// ---- DUTs/IO/PDOs/DRV_Target_position_05240F14.TcDUT
{attribute 'GeneratedUsingTerminal: EL7211-0010-0032'}
{attribute addProperty BoxType "EL7211-0010-0032"}
{attribute addProperty Id "Target_positionAT %Q*UDINT4"}
{attribute addProperty CRC "86249236"}
{attribute addProperty Size "4"}
TYPE DRV_Target_position_05240F14 EXTENDS TcoIo.OutputBase_10CEE7DE :
STRUCT
    {attribute addProperty Name "Target_position"}
    Target_position AT %Q* : UDINT;
END_STRUCT
END_TYPE

// ---- DUTs/IO/PDOs/InfoData_433F0777.TcDUT
{attribute 'GeneratedUsingTerminal: EL7211-0010-0032'}
{attribute addProperty BoxType "EL7211-0010-0032"}
{attribute addProperty Id "AdsAddrAT %I*TcoIo.TcoAmsAddr0DcOutputShiftAT %I*DINT4DcInputShiftAT %I*DINT4Chn0AT %I*USINT1Chn1AT %I*USINT1StateAT %I*UINT2"}
{attribute addProperty CRC "1128204151"}
{attribute addProperty Size "12"}
TYPE InfoData_433F0777 EXTENDS TcoIo.InputBase_8311D824 :
STRUCT
    {attribute addProperty Name "AdsAddr"}
    AdsAddr AT %I* : TcoIo.TcoAmsAddr;
    {attribute addProperty Name "DcOutputShift"}
    DcOutputShift AT %I* : DINT;
    {attribute addProperty Name "DcInputShift"}
    DcInputShift AT %I* : DINT;
    {attribute addProperty Name "Chn0"}
    Chn0 AT %I* : USINT;
    {attribute addProperty Name "Chn1"}
    Chn1 AT %I* : USINT;
    {attribute addProperty Name "State"}
    State AT %I* : UINT;
END_STRUCT
END_TYPE

// ---- DUTs/IO/PDOs/SAI_Inputs_Channel_9DCD6557.TcDUT
{attribute 'GeneratedUsingTerminal: EL3692-0000-0020'}
{attribute addProperty BoxType "EL3692-0000-0020"}
{attribute addProperty Id "StatusAT %I*Status_439F40C310ValueAT %I*DINT4"}
{attribute addProperty CRC "2647483735"}
{attribute addProperty Size "14"}
TYPE SAI_Inputs_Channel_9DCD6557 EXTENDS TcoIo.InputBase_8311D824 :
STRUCT
    {attribute addProperty Name "Status"}
    Status AT %I* : Status_439F40C3;
    {attribute addProperty Name "Value"}
    Value AT %I* : DINT;
END_STRUCT
END_TYPE

// ---- DUTs/IO/PDOs/SAI_Range_Channel_BDBF6DA9.TcDUT
{attribute 'GeneratedUsingTerminal: EL3692-0000-0020'}
{attribute addProperty BoxType "EL3692-0000-0020"}
{attribute addProperty Id "SettingsAT %I*Settings_24C049402"}
{attribute addProperty CRC "3183439273"}
{attribute addProperty Size "2"}
TYPE SAI_Range_Channel_BDBF6DA9 EXTENDS TcoIo.InputBase_8311D824 :
STRUCT
    {attribute addProperty Name "Settings"}
    Settings AT %I* : Settings_24C04940;
END_STRUCT
END_TYPE

// ---- DUTs/IO/PDOs/SAI_Inputs_Real_Channel_CCECF13D.TcDUT
{attribute 'GeneratedUsingTerminal: EL3692-0000-0020'}
{attribute addProperty BoxType "EL3692-0000-0020"}
{attribute addProperty Id "ValueAT %I*REAL4"}
{attribute addProperty CRC "3438080317"}
{attribute addProperty Size "4"}
TYPE SAI_Inputs_Real_Channel_CCECF13D EXTENDS TcoIo.InputBase_8311D824 :
STRUCT
    {attribute addProperty Name "Value"}
    Value AT %I* : REAL;
END_STRUCT
END_TYPE

// ---- DUTs/IO/PDOs/SAI_Range_Control_Channel_F5D9BC22.TcDUT
{attribute 'GeneratedUsingTerminal: EL3692-0000-0020'}
{attribute addProperty BoxType "EL3692-0000-0020"}
{attribute addProperty Id "ControlAT %Q*Control_E49DBA1B4"}
{attribute addProperty CRC "4124687394"}
{attribute addProperty Size "4"}
TYPE SAI_Range_Control_Channel_F5D9BC22 EXTENDS TcoIo.OutputBase_10CEE7DE :
STRUCT
    {attribute addProperty Name "Control"}
    Control AT %Q* : Control_E49DBA1B;
END_STRUCT
END_TYPE

// ---- DUTs/IO/PDOs/In_389F2F15.TcDUT
{attribute 'GeneratedUsingTerminal: Flexi Soft EtherCAT Gateway-0000-0001'}
{attribute addProperty BoxType "Flexi Soft EtherCAT Gateway-0000-0001"}
{attribute addProperty Id "DiagAT %I*USINT1In_Dataset1AT %I*ARRAY [0..9] OF BYTE0In_Dataset2AT %I*ARRAY [0..9] OF BYTE0In_Dataset3AT %I*ARRAY [0..9] OF BYTE0In_Dataset4AT %I*ARRAY [0..9] OF BYTE0In_Dataset5AT %I*ARRAY [0..9] OF BYTE0"}
{attribute addProperty CRC "949956373"}
{attribute addProperty Size "1"}
TYPE In_389F2F15 EXTENDS TcoIo.InputBase_8311D824 :
STRUCT
    {attribute addProperty Name "Diag"}
    Diag AT %I* : USINT;
    {attribute addProperty Name "In_Dataset1"}
    In_Dataset1 AT %I* : ARRAY[0..9] OF BYTE;
    {attribute addProperty Name "In_Dataset2"}
    In_Dataset2 AT %I* : ARRAY[0..9] OF BYTE;
    {attribute addProperty Name "In_Dataset3"}
    In_Dataset3 AT %I* : ARRAY[0..9] OF BYTE;
    {attribute addProperty Name "In_Dataset4"}
    In_Dataset4 AT %I* : ARRAY[0..9] OF BYTE;
    {attribute addProperty Name "In_Dataset5"}
    In_Dataset5 AT %I* : ARRAY[0..9] OF BYTE;
END_STRUCT
END_TYPE

// ---- DUTs/IO/PDOs/Out_81AAEF2D.TcDUT
{attribute 'GeneratedUsingTerminal: Flexi Soft EtherCAT Gateway-0000-0001'}
{attribute addProperty BoxType "Flexi Soft EtherCAT Gateway-0000-0001"}
{attribute addProperty Id "Out_Dataset1AT %Q*ARRAY [0..9] OF BYTE0Out_Dataset2AT %Q*ARRAY [0..9] OF BYTE0Out_Dataset3AT %Q*ARRAY [0..9] OF BYTE0Out_Dataset4AT %Q*ARRAY [0..9] OF BYTE0Out_Dataset5AT %Q*ARRAY [0..9] OF BYTE0"}
{attribute addProperty CRC "2175463213"}
{attribute addProperty Size "0"}
TYPE Out_81AAEF2D EXTENDS TcoIo.OutputBase_10CEE7DE :
STRUCT
    {attribute addProperty Name "Out_Dataset1"}
    Out_Dataset1 AT %Q* : ARRAY[0..9] OF BYTE;
    {attribute addProperty Name "Out_Dataset2"}
    Out_Dataset2 AT %Q* : ARRAY[0..9] OF BYTE;
    {attribute addProperty Name "Out_Dataset3"}
    Out_Dataset3 AT %Q* : ARRAY[0..9] OF BYTE;
    {attribute addProperty Name "Out_Dataset4"}
    Out_Dataset4 AT %Q* : ARRAY[0..9] OF BYTE;
    {attribute addProperty Name "Out_Dataset5"}
    Out_Dataset5 AT %Q* : ARRAY[0..9] OF BYTE;
END_STRUCT
END_TYPE

// ---- DUTs/IO/PDOs/ENC_Status_compact_4D066E1A.TcDUT
{attribute 'GeneratedUsingTerminal: EL7041-1000-0021'}
{attribute addProperty BoxType "EL7041-1000-0021"}
{attribute addProperty Id "StatusAT %I*Status_8CBE219F12Counter_valueAT %I*UINT2Latch_valueAT %I*UINT2"}
{attribute addProperty CRC "1292267034"}
{attribute addProperty Size "16"}
TYPE ENC_Status_compact_4D066E1A EXTENDS TcoIo.InputBase_8311D824 :
STRUCT
    {attribute addProperty Name "Status"}
    Status AT %I* : Status_8CBE219F;
    {attribute addProperty Name "Counter_value"}
    Counter_value AT %I* : UINT;
    {attribute addProperty Name "Latch_value"}
    Latch_value AT %I* : UINT;
END_STRUCT
END_TYPE

// ---- DUTs/IO/PDOs/STM_Status_36ED096F.TcDUT
{attribute 'GeneratedUsingTerminal: EL7041-1000-0021'}
{attribute addProperty BoxType "EL7041-1000-0021"}
{attribute addProperty Id "StatusAT %I*Status_B679584511"}
{attribute addProperty CRC "921504111"}
{attribute addProperty Size "11"}
TYPE STM_Status_36ED096F EXTENDS TcoIo.InputBase_8311D824 :
STRUCT
    {attribute addProperty Name "Status"}
    Status AT %I* : Status_B6795845;
END_STRUCT
END_TYPE

// ---- DUTs/IO/PDOs/ENC_Control_compact_21E2D14D.TcDUT
{attribute 'GeneratedUsingTerminal: EL7041-1000-0021'}
{attribute addProperty BoxType "EL7041-1000-0021"}
{attribute addProperty Id "ControlAT %Q*Control_6EF2C5D04Set_counter_valueAT %Q*UINT2"}
{attribute addProperty CRC "568512845"}
{attribute addProperty Size "6"}
TYPE ENC_Control_compact_21E2D14D EXTENDS TcoIo.OutputBase_10CEE7DE :
STRUCT
    {attribute addProperty Name "Control"}
    Control AT %Q* : Control_6EF2C5D0;
    {attribute addProperty Name "Set_counter_value"}
    Set_counter_value AT %Q* : UINT;
END_STRUCT
END_TYPE

// ---- DUTs/IO/PDOs/STM_Control_5A8B5016.TcDUT
{attribute 'GeneratedUsingTerminal: EL7041-1000-0021'}
{attribute addProperty BoxType "EL7041-1000-0021"}
{attribute addProperty Id "ControlAT %Q*Control_C948E0F23"}
{attribute addProperty CRC "1519079446"}
{attribute addProperty Size "3"}
TYPE STM_Control_5A8B5016 EXTENDS TcoIo.OutputBase_10CEE7DE :
STRUCT
    {attribute addProperty Name "Control"}
    Control AT %Q* : Control_C948E0F2;
END_STRUCT
END_TYPE

// ---- DUTs/IO/PDOs/STM_Velocity_A47A3F41.TcDUT
{attribute 'GeneratedUsingTerminal: EL7041-1000-0021'}
{attribute addProperty BoxType "EL7041-1000-0021"}
{attribute addProperty Id "VelocityAT %Q*INT2"}
{attribute addProperty CRC "2759475009"}
{attribute addProperty Size "2"}
TYPE STM_Velocity_A47A3F41 EXTENDS TcoIo.OutputBase_10CEE7DE :
STRUCT
    {attribute addProperty Name "Velocity"}
    Velocity AT %Q* : INT;
END_STRUCT
END_TYPE

// ---- DUTs/IO/PDOs/InfoData_D50C8545.TcDUT
{attribute 'GeneratedUsingTerminal: EL7041-1000-0021'}
{attribute addProperty BoxType "EL7041-1000-0021"}
{attribute addProperty Id "AdsAddrAT %I*TcoIo.TcoAmsAddr0Chn0AT %I*USINT1StateAT %I*UINT2"}
{attribute addProperty CRC "3574367557"}
{attribute addProperty Size "3"}
TYPE InfoData_D50C8545 EXTENDS TcoIo.InputBase_8311D824 :
STRUCT
    {attribute addProperty Name "AdsAddr"}
    AdsAddr AT %I* : TcoIo.TcoAmsAddr;
    {attribute addProperty Name "Chn0"}
    Chn0 AT %I* : USINT;
    {attribute addProperty Name "State"}
    State AT %I* : UINT;
END_STRUCT
END_TYPE

// ---- DUTs/IO/PDOs/AT_x_26CC547D.TcDUT
{attribute 'GeneratedUsingTerminal: IndraDrive MPB20-0003-0000'}
{attribute addProperty BoxType "IndraDrive MPB20-0003-0000"}
{attribute addProperty Id "Drive_status_wordAT %I*UINT2Position_feedback_value_1AT %I*DINT4"}
{attribute addProperty CRC "650925181"}
{attribute addProperty Size "6"}
TYPE AT_x_26CC547D EXTENDS TcoIo.InputBase_8311D824 :
STRUCT
    {attribute addProperty Name "Drive_status_word"}
    Drive_status_word AT %I* : UINT;
    {attribute addProperty Name "Position_feedback_value_1"}
    Position_feedback_value_1 AT %I* : DINT;
END_STRUCT
END_TYPE

// ---- DUTs/IO/Boxes/EK1200_013D0B49.TcDUT
{attribute 'GeneratedUsingTerminal: EK1200-1388-0000'}
{attribute addProperty VendorId "#x00000002"}
{attribute addProperty BoxType "EK1200-1388-0000"}
{attribute addProperty Description "EK1200-5000 EtherCAT Power supply (2A E-Bus)"}
{attribute addProperty Physics "YK"}
{attribute addProperty Id "EK1200"}
{attribute addProperty CRC "20777801"}
{attribute addProperty Size "0"}
TYPE EK1200_013D0B49 EXTENDS TcoIo.EtcSlaveBoxBase_77A0E4A7 :
STRUCT
END_STRUCT
END_TYPE

// ---- DUTs/IO/Boxes/EL6002_CD897635.TcDUT
{attribute 'GeneratedUsingTerminal: EL6002-0000-0019'}
{attribute addProperty VendorId "#x00000002"}
{attribute addProperty BoxType "EL6002-0000-0019"}
{attribute addProperty Description "EL6002 Interface 2Ch. (RS232)"}
{attribute addProperty Physics "KK"}
{attribute addProperty Id "COM_TxPDO_Map_Inputs_Channel_1AT %I*COM_TxPDO_Map_Inputs_Channel_3801C95E30COM_TxPDO_Map_Inputs_Channel_2AT %I*COM_TxPDO_Map_Inputs_Channel_3801C95E30COM_RxPDO_Map_Outputs_Channel_1AT %Q*COM_RxPDO_Map_Outputs_Channel_EADA2E0D27COM_RxPDO_Map_Outputs_Channel_2AT %Q*COM_RxPDO_Map_Outputs_Channel_EADA2E0D27WcStateAT %I*WcState_9091E0EB2InfoDataAT %I*InfoData_23CBA8372"}
{attribute addProperty CRC "3448337973"}
{attribute addProperty Size "118"}
TYPE EL6002_CD897635 EXTENDS TcoIo.EtcSlaveTerminalBase_947E5A46 :
STRUCT
    {attribute addProperty Name "COM_TxPDO_Map_Inputs_Channel_1"}
    COM_TxPDO_Map_Inputs_Channel_1 : COM_TxPDO_Map_Inputs_Channel_3801C95E;
    {attribute addProperty Name "COM_TxPDO_Map_Inputs_Channel_2"}
    COM_TxPDO_Map_Inputs_Channel_2 : COM_TxPDO_Map_Inputs_Channel_3801C95E;
    {attribute addProperty Name "COM_RxPDO_Map_Outputs_Channel_1"}
    COM_RxPDO_Map_Outputs_Channel_1 : COM_RxPDO_Map_Outputs_Channel_EADA2E0D;
    {attribute addProperty Name "COM_RxPDO_Map_Outputs_Channel_2"}
    COM_RxPDO_Map_Outputs_Channel_2 : COM_RxPDO_Map_Outputs_Channel_EADA2E0D;
    {attribute addProperty Name "WcState"}
    WcState : TcoIo.WcState_9091E0EB;
    {attribute addProperty Name "InfoData"}
    InfoData : TcoIo.InfoData_23CBA837;
END_STRUCT
END_TYPE

// ---- DUTs/IO/Boxes/EL1809_32157CFD.TcDUT
{attribute 'GeneratedUsingTerminal: EL1809-0000-0018'}
{attribute addProperty VendorId "#x00000002"}
{attribute addProperty BoxType "EL1809-0000-0018"}
{attribute addProperty Description "EL1809 16Ch. Dig. Input 24V, 3ms"}
{attribute addProperty Physics "KK"}
{attribute addProperty Id "Channel_1AT %I*Channel_830843C11Channel_2AT %I*Channel_830843C11Channel_3AT %I*Channel_830843C11Channel_4AT %I*Channel_830843C11Channel_5AT %I*Channel_830843C11Channel_6AT %I*Channel_830843C11Channel_7AT %I*Channel_830843C11Channel_8AT %I*Channel_830843C11Channel_9AT %I*Channel_830843C11Channel_10AT %I*Channel_830843C11Channel_11AT %I*Channel_830843C11Channel_12AT %I*Channel_830843C11Channel_13AT %I*Channel_830843C11Channel_14AT %I*Channel_830843C11Channel_15AT %I*Channel_830843C11Channel_16AT %I*Channel_830843C11WcStateAT %I*WcState_9091E0EB2InfoDataAT %I*InfoData_6F19DB2B2"}
{attribute addProperty CRC "840269053"}
{attribute addProperty Size "20"}
TYPE EL1809_32157CFD EXTENDS TcoIo.EtcSlaveTerminalBase_947E5A46 :
STRUCT
    {attribute addProperty Name "Channel_1"}
    Channel_1 : Channel_830843C1;
    {attribute addProperty Name "Channel_2"}
    Channel_2 : Channel_830843C1;
    {attribute addProperty Name "Channel_3"}
    Channel_3 : Channel_830843C1;
    {attribute addProperty Name "Channel_4"}
    Channel_4 : Channel_830843C1;
    {attribute addProperty Name "Channel_5"}
    Channel_5 : Channel_830843C1;
    {attribute addProperty Name "Channel_6"}
    Channel_6 : Channel_830843C1;
    {attribute addProperty Name "Channel_7"}
    Channel_7 : Channel_830843C1;
    {attribute addProperty Name "Channel_8"}
    Channel_8 : Channel_830843C1;
    {attribute addProperty Name "Channel_9"}
    Channel_9 : Channel_830843C1;
    {attribute addProperty Name "Channel_10"}
    Channel_10 : Channel_830843C1;
    {attribute addProperty Name "Channel_11"}
    Channel_11 : Channel_830843C1;
    {attribute addProperty Name "Channel_12"}
    Channel_12 : Channel_830843C1;
    {attribute addProperty Name "Channel_13"}
    Channel_13 : Channel_830843C1;
    {attribute addProperty Name "Channel_14"}
    Channel_14 : Channel_830843C1;
    {attribute addProperty Name "Channel_15"}
    Channel_15 : Channel_830843C1;
    {attribute addProperty Name "Channel_16"}
    Channel_16 : Channel_830843C1;
    {attribute addProperty Name "WcState"}
    WcState : TcoIo.WcState_9091E0EB;
    {attribute addProperty Name "InfoData"}
    InfoData : TcoIo.InfoData_6F19DB2B;
END_STRUCT
END_TYPE

// ---- DUTs/IO/Boxes/EL2809_2B6483BD.TcDUT
{attribute 'GeneratedUsingTerminal: EL2809-0000-0018'}
{attribute addProperty VendorId "#x00000002"}
{attribute addProperty BoxType "EL2809-0000-0018"}
{attribute addProperty Description "EL2809 16Ch. Dig. Output 24V, 0.5A"}
{attribute addProperty Physics "KK"}
{attribute addProperty Id "Channel_1AT %Q*Channel_42CA91F71Channel_2AT %Q*Channel_42CA91F71Channel_3AT %Q*Channel_42CA91F71Channel_4AT %Q*Channel_42CA91F71Channel_5AT %Q*Channel_42CA91F71Channel_6AT %Q*Channel_42CA91F71Channel_7AT %Q*Channel_42CA91F71Channel_8AT %Q*Channel_42CA91F71Channel_9AT %Q*Channel_42CA91F71Channel_10AT %Q*Channel_42CA91F71Channel_11AT %Q*Channel_42CA91F71Channel_12AT %Q*Channel_42CA91F71Channel_13AT %Q*Channel_42CA91F71Channel_14AT %Q*Channel_42CA91F71Channel_15AT %Q*Channel_42CA91F71Channel_16AT %Q*Channel_42CA91F71WcStateAT %I*WcState_0B2B16F91InfoDataAT %I*InfoData_6F19DB2B2"}
{attribute addProperty CRC "728007613"}
{attribute addProperty Size "19"}
TYPE EL2809_2B6483BD EXTENDS TcoIo.EtcSlaveTerminalBase_947E5A46 :
STRUCT
    {attribute addProperty Name "Channel_1"}
    Channel_1 : Channel_42CA91F7;
    {attribute addProperty Name "Channel_2"}
    Channel_2 : Channel_42CA91F7;
    {attribute addProperty Name "Channel_3"}
    Channel_3 : Channel_42CA91F7;
    {attribute addProperty Name "Channel_4"}
    Channel_4 : Channel_42CA91F7;
    {attribute addProperty Name "Channel_5"}
    Channel_5 : Channel_42CA91F7;
    {attribute addProperty Name "Channel_6"}
    Channel_6 : Channel_42CA91F7;
    {attribute addProperty Name "Channel_7"}
    Channel_7 : Channel_42CA91F7;
    {attribute addProperty Name "Channel_8"}
    Channel_8 : Channel_42CA91F7;
    {attribute addProperty Name "Channel_9"}
    Channel_9 : Channel_42CA91F7;
    {attribute addProperty Name "Channel_10"}
    Channel_10 : Channel_42CA91F7;
    {attribute addProperty Name "Channel_11"}
    Channel_11 : Channel_42CA91F7;
    {attribute addProperty Name "Channel_12"}
    Channel_12 : Channel_42CA91F7;
    {attribute addProperty Name "Channel_13"}
    Channel_13 : Channel_42CA91F7;
    {attribute addProperty Name "Channel_14"}
    Channel_14 : Channel_42CA91F7;
    {attribute addProperty Name "Channel_15"}
    Channel_15 : Channel_42CA91F7;
    {attribute addProperty Name "Channel_16"}
    Channel_16 : Channel_42CA91F7;
    {attribute addProperty Name "WcState"}
    WcState : TcoIo.WcState_0B2B16F9;
    {attribute addProperty Name "InfoData"}
    InfoData : TcoIo.InfoData_6F19DB2B;
END_STRUCT
END_TYPE

// ---- DUTs/IO/Boxes/EL4004_E203F875.TcDUT
{attribute 'GeneratedUsingTerminal: EL4004-0000-0020'}
{attribute addProperty VendorId "#x00000002"}
{attribute addProperty BoxType "EL4004-0000-0020"}
{attribute addProperty Description "EL4004 4Ch. Ana. Output 0-10V, 12bit"}
{attribute addProperty Physics "KK"}
{attribute addProperty Id "AO_Outputs_Channel_1AT %Q*AO_Output_Channel_BA7EBB7C2AO_Outputs_Channel_2AT %Q*AO_Output_Channel_BA7EBB7C2AO_Outputs_Channel_3AT %Q*AO_Output_Channel_BA7EBB7C2AO_Outputs_Channel_4AT %Q*AO_Output_Channel_BA7EBB7C2WcStateAT %I*WcState_0B2B16F91InfoDataAT %I*InfoData_23CBA8372"}
{attribute addProperty CRC "3791911029"}
{attribute addProperty Size "11"}
TYPE EL4004_E203F875 EXTENDS TcoIo.EtcSlaveTerminalBase_947E5A46 :
STRUCT
    {attribute addProperty Name "AO_Outputs_Channel_1"}
    AO_Outputs_Channel_1 : AO_Output_Channel_BA7EBB7C;
    {attribute addProperty Name "AO_Outputs_Channel_2"}
    AO_Outputs_Channel_2 : AO_Output_Channel_BA7EBB7C;
    {attribute addProperty Name "AO_Outputs_Channel_3"}
    AO_Outputs_Channel_3 : AO_Output_Channel_BA7EBB7C;
    {attribute addProperty Name "AO_Outputs_Channel_4"}
    AO_Outputs_Channel_4 : AO_Output_Channel_BA7EBB7C;
    {attribute addProperty Name "WcState"}
    WcState : TcoIo.WcState_0B2B16F9;
    {attribute addProperty Name "InfoData"}
    InfoData : TcoIo.InfoData_23CBA837;
END_STRUCT
END_TYPE

// ---- DUTs/IO/Boxes/EL6001_0DE01E7E.TcDUT
{attribute 'GeneratedUsingTerminal: EL6001-0000-0020'}
{attribute addProperty VendorId "#x00000002"}
{attribute addProperty BoxType "EL6001-0000-0020"}
{attribute addProperty Description "EL6001 Interface (RS232)"}
{attribute addProperty Physics "KK"}
{attribute addProperty Id "COM_InputsAT %I*COM_Inputs_3801C95E30COM_OutputsAT %Q*COM_Outputs_DEF408EC27WcStateAT %I*WcState_9091E0EB2InfoDataAT %I*InfoData_23CBA8372"}
{attribute addProperty CRC "232791678"}
{attribute addProperty Size "61"}
TYPE EL6001_0DE01E7E EXTENDS TcoIo.EtcSlaveTerminalBase_947E5A46 :
STRUCT
    {attribute addProperty Name "COM_Inputs"}
    COM_Inputs : COM_Inputs_3801C95E;
    {attribute addProperty Name "COM_Outputs"}
    COM_Outputs : COM_Outputs_DEF408EC;
    {attribute addProperty Name "WcState"}
    WcState : TcoIo.WcState_9091E0EB;
    {attribute addProperty Name "InfoData"}
    InfoData : TcoIo.InfoData_23CBA837;
END_STRUCT
END_TYPE

// ---- DUTs/IO/Boxes/EL9011_D65D3D32.TcDUT
{attribute 'GeneratedUsingTerminal: EL9011--0000'}
{attribute addProperty VendorId "#x00000002"}
{attribute addProperty BoxType "EL9011--0000"}
{attribute addProperty Description "EL9011 End Terminal"}
{attribute addProperty Physics ""}
{attribute addProperty Id "EL9011"}
{attribute addProperty CRC "3596434738"}
{attribute addProperty Size "0"}
TYPE EL9011_D65D3D32 EXTENDS TcoIo.EtcSlaveEndTerminalBase_866C7F0C :
STRUCT
END_STRUCT
END_TYPE

// ---- DUTs/IO/Boxes/EK1100_1FC0878B.TcDUT
{attribute 'GeneratedUsingTerminal: EK1100-0000-0018'}
{attribute addProperty VendorId "#x00000002"}
{attribute addProperty BoxType "EK1100-0000-0018"}
{attribute addProperty Description "EK1100 EtherCAT Coupler (2A E-Bus)"}
{attribute addProperty Physics "YKY"}
{attribute addProperty Id "InfoDataAT %I*InfoData_6F19DB2B2"}
{attribute addProperty CRC "532711307"}
{attribute addProperty Size "2"}
TYPE EK1100_1FC0878B EXTENDS TcoIo.EtcSlaveBoxBase_77A0E4A7 :
STRUCT
    {attribute addProperty Name "InfoData"}
    InfoData : TcoIo.InfoData_6F19DB2B;
END_STRUCT
END_TYPE

// ---- DUTs/IO/Boxes/EK1122_1FC0878B.TcDUT
{attribute 'GeneratedUsingTerminal: EK1122-0000-0018'}
{attribute addProperty VendorId "#x00000002"}
{attribute addProperty BoxType "EK1122-0000-0018"}
{attribute addProperty Description "EK1122 2 port EtherCAT junction"}
{attribute addProperty Physics "KYKY"}
{attribute addProperty Id "InfoDataAT %I*InfoData_6F19DB2B2"}
{attribute addProperty CRC "532711307"}
{attribute addProperty Size "2"}
TYPE EK1122_1FC0878B EXTENDS TcoIo.EtcSlaveTerminalBase_947E5A46 :
STRUCT
    {attribute addProperty Name "InfoData"}
    InfoData : TcoIo.InfoData_6F19DB2B;
END_STRUCT
END_TYPE

// ---- DUTs/IO/Boxes/EL3174_B71BFF42.TcDUT
{attribute 'GeneratedUsingTerminal: EL3174-0002-0017'}
{attribute addProperty VendorId "#x00000002"}
{attribute addProperty BoxType "EL3174-0002-0017"}
{attribute addProperty Description "EL3174-0002 4Ch. Ana. Input +/-10V, +/-20mA 16 Bit, Isolated Channels"}
{attribute addProperty Physics "KK"}
{attribute addProperty Id "AI_Standard_Channel_1AT %I*AI_Standard_Channel_A8DF64E310AI_Standard_Channel_2AT %I*AI_Standard_Channel_A8DF64E310AI_Standard_Channel_3AT %I*AI_Standard_Channel_A8DF64E310AI_Standard_Channel_4AT %I*AI_Standard_Channel_A8DF64E310WcStateAT %I*WcState_9091E0EB2InfoDataAT %I*InfoData_23CBA8372"}
{attribute addProperty CRC "3072065346"}
{attribute addProperty Size "44"}
TYPE EL3174_B71BFF42 EXTENDS TcoIo.EtcSlaveTerminalBase_947E5A46 :
STRUCT
    {attribute addProperty Name "AI_Standard_Channel_1"}
    AI_Standard_Channel_1 : AI_Standard_Channel_A8DF64E3;
    {attribute addProperty Name "AI_Standard_Channel_2"}
    AI_Standard_Channel_2 : AI_Standard_Channel_A8DF64E3;
    {attribute addProperty Name "AI_Standard_Channel_3"}
    AI_Standard_Channel_3 : AI_Standard_Channel_A8DF64E3;
    {attribute addProperty Name "AI_Standard_Channel_4"}
    AI_Standard_Channel_4 : AI_Standard_Channel_A8DF64E3;
    {attribute addProperty Name "WcState"}
    WcState : TcoIo.WcState_9091E0EB;
    {attribute addProperty Name "InfoData"}
    InfoData : TcoIo.InfoData_23CBA837;
END_STRUCT
END_TYPE

// ---- DUTs/IO/Boxes/EL3011_7A495228.TcDUT
{attribute 'GeneratedUsingTerminal: EL3011-0000-0018'}
{attribute addProperty VendorId "#x00000002"}
{attribute addProperty BoxType "EL3011-0000-0018"}
{attribute addProperty Description "EL3011 4Ch. Ana. Input 0-20mA DIFF"}
{attribute addProperty Physics "KK"}
{attribute addProperty Id "AI_StandardAT %I*AI_Standard_Channel_4A3944819WcStateAT %I*WcState_9091E0EB2InfoDataAT %I*InfoData_23CBA8372"}
{attribute addProperty CRC "2051625512"}
{attribute addProperty Size "13"}
TYPE EL3011_7A495228 EXTENDS TcoIo.EtcSlaveTerminalBase_947E5A46 :
STRUCT
    {attribute addProperty Name "AI_Standard"}
    AI_Standard : AI_Standard_Channel_4A394481;
    {attribute addProperty Name "WcState"}
    WcState : TcoIo.WcState_9091E0EB;
    {attribute addProperty Name "InfoData"}
    InfoData : TcoIo.InfoData_23CBA837;
END_STRUCT
END_TYPE

// ---- DUTs/IO/Boxes/EL2008_E2806B95.TcDUT
{attribute 'GeneratedUsingTerminal: EL2008-0000-0017'}
{attribute addProperty VendorId "#x00000002"}
{attribute addProperty BoxType "EL2008-0000-0017"}
{attribute addProperty Description "EL2008 8Ch. Dig. Output 24V, 0.5A"}
{attribute addProperty Physics "KK"}
{attribute addProperty Id "Channel_1AT %Q*Channel_42CA91F71Channel_2AT %Q*Channel_42CA91F71Channel_3AT %Q*Channel_42CA91F71Channel_4AT %Q*Channel_42CA91F71Channel_5AT %Q*Channel_42CA91F71Channel_6AT %Q*Channel_42CA91F71Channel_7AT %Q*Channel_42CA91F71Channel_8AT %Q*Channel_42CA91F71WcStateAT %I*WcState_0B2B16F91InfoDataAT %I*InfoData_6F19DB2B2"}
{attribute addProperty CRC "3800066965"}
{attribute addProperty Size "11"}
TYPE EL2008_E2806B95 EXTENDS TcoIo.EtcSlaveTerminalBase_947E5A46 :
STRUCT
    {attribute addProperty Name "Channel_1"}
    Channel_1 : Channel_42CA91F7;
    {attribute addProperty Name "Channel_2"}
    Channel_2 : Channel_42CA91F7;
    {attribute addProperty Name "Channel_3"}
    Channel_3 : Channel_42CA91F7;
    {attribute addProperty Name "Channel_4"}
    Channel_4 : Channel_42CA91F7;
    {attribute addProperty Name "Channel_5"}
    Channel_5 : Channel_42CA91F7;
    {attribute addProperty Name "Channel_6"}
    Channel_6 : Channel_42CA91F7;
    {attribute addProperty Name "Channel_7"}
    Channel_7 : Channel_42CA91F7;
    {attribute addProperty Name "Channel_8"}
    Channel_8 : Channel_42CA91F7;
    {attribute addProperty Name "WcState"}
    WcState : TcoIo.WcState_0B2B16F9;
    {attribute addProperty Name "InfoData"}
    InfoData : TcoIo.InfoData_6F19DB2B;
END_STRUCT
END_TYPE

// ---- DUTs/IO/Boxes/EK1110_1FC0878B.TcDUT
{attribute 'GeneratedUsingTerminal: EK1110-0000-0017'}
{attribute addProperty VendorId "#x00000002"}
{attribute addProperty BoxType "EK1110-0000-0017"}
{attribute addProperty Description "EK1110 EtherCAT extension"}
{attribute addProperty Physics "KY"}
{attribute addProperty Id "InfoDataAT %I*InfoData_6F19DB2B2"}
{attribute addProperty CRC "532711307"}
{attribute addProperty Size "2"}
TYPE EK1110_1FC0878B EXTENDS TcoIo.EtcSlaveTerminalBase_947E5A46 :
STRUCT
    {attribute addProperty Name "InfoData"}
    InfoData : TcoIo.InfoData_6F19DB2B;
END_STRUCT
END_TYPE

// ---- DUTs/IO/Boxes/EL1819_32157CFD.TcDUT
{attribute 'GeneratedUsingTerminal: EL1819-0000-0018'}
{attribute addProperty VendorId "#x00000002"}
{attribute addProperty BoxType "EL1819-0000-0018"}
{attribute addProperty Description "EL1819 16Ch. Dig. Input 24V, 10Ã‚Âµs"}
{attribute addProperty Physics "KK"}
{attribute addProperty Id "Channel_1AT %I*Channel_830843C11Channel_2AT %I*Channel_830843C11Channel_3AT %I*Channel_830843C11Channel_4AT %I*Channel_830843C11Channel_5AT %I*Channel_830843C11Channel_6AT %I*Channel_830843C11Channel_7AT %I*Channel_830843C11Channel_8AT %I*Channel_830843C11Channel_9AT %I*Channel_830843C11Channel_10AT %I*Channel_830843C11Channel_11AT %I*Channel_830843C11Channel_12AT %I*Channel_830843C11Channel_13AT %I*Channel_830843C11Channel_14AT %I*Channel_830843C11Channel_15AT %I*Channel_830843C11Channel_16AT %I*Channel_830843C11WcStateAT %I*WcState_9091E0EB2InfoDataAT %I*InfoData_6F19DB2B2"}
{attribute addProperty CRC "840269053"}
{attribute addProperty Size "20"}
TYPE EL1819_32157CFD EXTENDS TcoIo.EtcSlaveTerminalBase_947E5A46 :
STRUCT
    {attribute addProperty Name "Channel_1"}
    Channel_1 : Channel_830843C1;
    {attribute addProperty Name "Channel_2"}
    Channel_2 : Channel_830843C1;
    {attribute addProperty Name "Channel_3"}
    Channel_3 : Channel_830843C1;
    {attribute addProperty Name "Channel_4"}
    Channel_4 : Channel_830843C1;
    {attribute addProperty Name "Channel_5"}
    Channel_5 : Channel_830843C1;
    {attribute addProperty Name "Channel_6"}
    Channel_6 : Channel_830843C1;
    {attribute addProperty Name "Channel_7"}
    Channel_7 : Channel_830843C1;
    {attribute addProperty Name "Channel_8"}
    Channel_8 : Channel_830843C1;
    {attribute addProperty Name "Channel_9"}
    Channel_9 : Channel_830843C1;
    {attribute addProperty Name "Channel_10"}
    Channel_10 : Channel_830843C1;
    {attribute addProperty Name "Channel_11"}
    Channel_11 : Channel_830843C1;
    {attribute addProperty Name "Channel_12"}
    Channel_12 : Channel_830843C1;
    {attribute addProperty Name "Channel_13"}
    Channel_13 : Channel_830843C1;
    {attribute addProperty Name "Channel_14"}
    Channel_14 : Channel_830843C1;
    {attribute addProperty Name "Channel_15"}
    Channel_15 : Channel_830843C1;
    {attribute addProperty Name "Channel_16"}
    Channel_16 : Channel_830843C1;
    {attribute addProperty Name "WcState"}
    WcState : TcoIo.WcState_9091E0EB;
    {attribute addProperty Name "InfoData"}
    InfoData : TcoIo.InfoData_6F19DB2B;
END_STRUCT
END_TYPE

// ---- DUTs/IO/Boxes/EL2788_E2806B95.TcDUT
{attribute 'GeneratedUsingTerminal: EL2788-0000-0016'}
{attribute addProperty VendorId "#x00000002"}
{attribute addProperty BoxType "EL2788-0000-0016"}
{attribute addProperty Description "EL2788 8Ch. Dig. Output 24V AC/DC, 2A"}
{attribute addProperty Physics "KK"}
{attribute addProperty Id "Channel_1AT %Q*Channel_42CA91F71Channel_2AT %Q*Channel_42CA91F71Channel_3AT %Q*Channel_42CA91F71Channel_4AT %Q*Channel_42CA91F71Channel_5AT %Q*Channel_42CA91F71Channel_6AT %Q*Channel_42CA91F71Channel_7AT %Q*Channel_42CA91F71Channel_8AT %Q*Channel_42CA91F71WcStateAT %I*WcState_0B2B16F91InfoDataAT %I*InfoData_6F19DB2B2"}
{attribute addProperty CRC "3800066965"}
{attribute addProperty Size "11"}
TYPE EL2788_E2806B95 EXTENDS TcoIo.EtcSlaveTerminalBase_947E5A46 :
STRUCT
    {attribute addProperty Name "Channel_1"}
    Channel_1 : Channel_42CA91F7;
    {attribute addProperty Name "Channel_2"}
    Channel_2 : Channel_42CA91F7;
    {attribute addProperty Name "Channel_3"}
    Channel_3 : Channel_42CA91F7;
    {attribute addProperty Name "Channel_4"}
    Channel_4 : Channel_42CA91F7;
    {attribute addProperty Name "Channel_5"}
    Channel_5 : Channel_42CA91F7;
    {attribute addProperty Name "Channel_6"}
    Channel_6 : Channel_42CA91F7;
    {attribute addProperty Name "Channel_7"}
    Channel_7 : Channel_42CA91F7;
    {attribute addProperty Name "Channel_8"}
    Channel_8 : Channel_42CA91F7;
    {attribute addProperty Name "WcState"}
    WcState : TcoIo.WcState_0B2B16F9;
    {attribute addProperty Name "InfoData"}
    InfoData : TcoIo.InfoData_6F19DB2B;
END_STRUCT
END_TYPE

// ---- DUTs/IO/Boxes/EL3773_F128CC82.TcDUT
{attribute 'GeneratedUsingTerminal: EL3773-0000-0021'}
{attribute addProperty VendorId "#x00000002"}
{attribute addProperty BoxType "EL3773-0000-0021"}
{attribute addProperty Description "EL3773 3 Ch. Power Monitoring, Oversample"}
{attribute addProperty Physics "KK"}
{attribute addProperty Id "L1_Voltage_StatusAT %I*L1_Voltage_Status_7371B0437L1_Voltage_SamplesAT %I*L1_Voltage_Samples_41AEB7FF20L1_Current_StatusAT %I*L1_Current_Status_82DECBF67L1_Current_SamplesAT %I*L1_Current_Samples_9EC08B3E20L2_Voltage_StatusAT %I*L2_Voltage_Status_0D1813FE7L2_Voltage_SamplesAT %I*L2_Voltage_Samples_75D833AF20L2_Current_StatusAT %I*L2_Current_Status_FCB7684B7L2_Current_SamplesAT %I*L2_Current_Samples_AAB60F6E20L3_Voltage_StatusAT %I*L3_Voltage_Status_273F72957L3_Voltage_SamplesAT %I*L3_Voltage_Samples_660A4F9F20L3_Current_StatusAT %I*L3_Current_Status_D69009207L3_Current_SamplesAT %I*L3_Current_Samples_B964735E20AI_NextSync1TimeAT %I*AI_NextSync1Time_6DC4D2968AI_Sample_CountAT %I*AI_Sample_Count_EA88CAD92WcStateAT %I*WcState_9091E0EB2InfoDataAT %I*InfoData_B84DBEC510"}
{attribute addProperty CRC "4045982850"}
{attribute addProperty Size "184"}
TYPE EL3773_F128CC82 EXTENDS TcoIo.EtcSlaveTerminalBase_947E5A46 :
STRUCT
    {attribute addProperty Name "L1_Voltage_Status"}
    L1_Voltage_Status : L1_Voltage_Status_7371B043;
    {attribute addProperty Name "L1_Voltage_Samples"}
    L1_Voltage_Samples : L1_Voltage_Samples_41AEB7FF;
    {attribute addProperty Name "L1_Current_Status"}
    L1_Current_Status : L1_Current_Status_82DECBF6;
    {attribute addProperty Name "L1_Current_Samples"}
    L1_Current_Samples : L1_Current_Samples_9EC08B3E;
    {attribute addProperty Name "L2_Voltage_Status"}
    L2_Voltage_Status : L2_Voltage_Status_0D1813FE;
    {attribute addProperty Name "L2_Voltage_Samples"}
    L2_Voltage_Samples : L2_Voltage_Samples_75D833AF;
    {attribute addProperty Name "L2_Current_Status"}
    L2_Current_Status : L2_Current_Status_FCB7684B;
    {attribute addProperty Name "L2_Current_Samples"}
    L2_Current_Samples : L2_Current_Samples_AAB60F6E;
    {attribute addProperty Name "L3_Voltage_Status"}
    L3_Voltage_Status : L3_Voltage_Status_273F7295;
    {attribute addProperty Name "L3_Voltage_Samples"}
    L3_Voltage_Samples : L3_Voltage_Samples_660A4F9F;
    {attribute addProperty Name "L3_Current_Status"}
    L3_Current_Status : L3_Current_Status_D6900920;
    {attribute addProperty Name "L3_Current_Samples"}
    L3_Current_Samples : L3_Current_Samples_B964735E;
    {attribute addProperty Name "AI_NextSync1Time"}
    AI_NextSync1Time : AI_NextSync1Time_6DC4D296;
    {attribute addProperty Name "AI_Sample_Count"}
    AI_Sample_Count : AI_Sample_Count_EA88CAD9;
    {attribute addProperty Name "WcState"}
    WcState : TcoIo.WcState_9091E0EB;
    {attribute addProperty Name "InfoData"}
    InfoData : InfoData_B84DBEC5;
END_STRUCT
END_TYPE

// ---- DUTs/IO/Boxes/EL2258_E3B260FA.TcDUT
{attribute 'GeneratedUsingTerminal: EL2258-0000-0017'}
{attribute addProperty VendorId "#x00000002"}
{attribute addProperty BoxType "EL2258-0000-0017"}
{attribute addProperty Description "EL2258 8Ch. Dig Output 24V with Multi-Time-Stamp"}
{attribute addProperty Physics "KK"}
{attribute addProperty Id "MTO_Inputs_Channel_1AT %I*MTO_Inputs_Channel_53C09E8B6MTO_Inputs_Channel_2AT %I*MTO_Inputs_Channel_53C09E8B6MTO_Inputs_Channel_3AT %I*MTO_Inputs_Channel_53C09E8B6MTO_Inputs_Channel_4AT %I*MTO_Inputs_Channel_53C09E8B6MTO_Inputs_Channel_5AT %I*MTO_Inputs_Channel_53C09E8B6MTO_Inputs_Channel_6AT %I*MTO_Inputs_Channel_53C09E8B6MTO_Inputs_Channel_7AT %I*MTO_Inputs_Channel_53C09E8B6MTO_Inputs_Channel_8AT %I*MTO_Inputs_Channel_53C09E8B6MTO_Outputs_10x_Channel_1AT %Q*MTO_Outputs_10x_Channel_A3C0C02256MTO_Outputs_10x_Channel_2AT %Q*MTO_Outputs_10x_Channel_A3C0C02256MTO_Outputs_10x_Channel_3AT %Q*MTO_Outputs_10x_Channel_A3C0C02256MTO_Outputs_10x_Channel_4AT %Q*MTO_Outputs_10x_Channel_A3C0C02256MTO_Outputs_10x_Channel_5AT %Q*MTO_Outputs_10x_Channel_A3C0C02256MTO_Outputs_10x_Channel_6AT %Q*MTO_Outputs_10x_Channel_A3C0C02256MTO_Outputs_10x_Channel_7AT %Q*MTO_Outputs_10x_Channel_A3C0C02256MTO_Outputs_10x_Channel_8AT %Q*MTO_Outputs_10x_Channel_A3C0C02256WcStateAT %I*WcState_9091E0EB2InfoDataAT %I*InfoData_B84DBEC510"}
{attribute addProperty CRC "3820118266"}
{attribute addProperty Size "508"}
TYPE EL2258_E3B260FA EXTENDS TcoIo.EtcSlaveTerminalBase_947E5A46 :
STRUCT
    {attribute addProperty Name "MTO_Inputs_Channel_1"}
    MTO_Inputs_Channel_1 : MTO_Inputs_Channel_53C09E8B;
    {attribute addProperty Name "MTO_Inputs_Channel_2"}
    MTO_Inputs_Channel_2 : MTO_Inputs_Channel_53C09E8B;
    {attribute addProperty Name "MTO_Inputs_Channel_3"}
    MTO_Inputs_Channel_3 : MTO_Inputs_Channel_53C09E8B;
    {attribute addProperty Name "MTO_Inputs_Channel_4"}
    MTO_Inputs_Channel_4 : MTO_Inputs_Channel_53C09E8B;
    {attribute addProperty Name "MTO_Inputs_Channel_5"}
    MTO_Inputs_Channel_5 : MTO_Inputs_Channel_53C09E8B;
    {attribute addProperty Name "MTO_Inputs_Channel_6"}
    MTO_Inputs_Channel_6 : MTO_Inputs_Channel_53C09E8B;
    {attribute addProperty Name "MTO_Inputs_Channel_7"}
    MTO_Inputs_Channel_7 : MTO_Inputs_Channel_53C09E8B;
    {attribute addProperty Name "MTO_Inputs_Channel_8"}
    MTO_Inputs_Channel_8 : MTO_Inputs_Channel_53C09E8B;
    {attribute addProperty Name "MTO_Outputs_10x_Channel_1"}
    MTO_Outputs_10x_Channel_1 : MTO_Outputs_10x_Channel_A3C0C022;
    {attribute addProperty Name "MTO_Outputs_10x_Channel_2"}
    MTO_Outputs_10x_Channel_2 : MTO_Outputs_10x_Channel_A3C0C022;
    {attribute addProperty Name "MTO_Outputs_10x_Channel_3"}
    MTO_Outputs_10x_Channel_3 : MTO_Outputs_10x_Channel_A3C0C022;
    {attribute addProperty Name "MTO_Outputs_10x_Channel_4"}
    MTO_Outputs_10x_Channel_4 : MTO_Outputs_10x_Channel_A3C0C022;
    {attribute addProperty Name "MTO_Outputs_10x_Channel_5"}
    MTO_Outputs_10x_Channel_5 : MTO_Outputs_10x_Channel_A3C0C022;
    {attribute addProperty Name "MTO_Outputs_10x_Channel_6"}
    MTO_Outputs_10x_Channel_6 : MTO_Outputs_10x_Channel_A3C0C022;
    {attribute addProperty Name "MTO_Outputs_10x_Channel_7"}
    MTO_Outputs_10x_Channel_7 : MTO_Outputs_10x_Channel_A3C0C022;
    {attribute addProperty Name "MTO_Outputs_10x_Channel_8"}
    MTO_Outputs_10x_Channel_8 : MTO_Outputs_10x_Channel_A3C0C022;
    {attribute addProperty Name "WcState"}
    WcState : TcoIo.WcState_9091E0EB;
    {attribute addProperty Name "InfoData"}
    InfoData : InfoData_B84DBEC5;
END_STRUCT
END_TYPE

// ---- DUTs/IO/Boxes/EL3164_B71BFF42.TcDUT
{attribute 'GeneratedUsingTerminal: EL3164-0000-0020'}
{attribute addProperty VendorId "#x00000002"}
{attribute addProperty BoxType "EL3164-0000-0020"}
{attribute addProperty Description "EL3164 4Ch. Ana. Input 0-10V"}
{attribute addProperty Physics "KK"}
{attribute addProperty Id "AI_Standard_Channel_1AT %I*AI_Standard_Channel_A8DF64E310AI_Standard_Channel_2AT %I*AI_Standard_Channel_A8DF64E310AI_Standard_Channel_3AT %I*AI_Standard_Channel_A8DF64E310AI_Standard_Channel_4AT %I*AI_Standard_Channel_A8DF64E310WcStateAT %I*WcState_9091E0EB2InfoDataAT %I*InfoData_23CBA8372"}
{attribute addProperty CRC "3072065346"}
{attribute addProperty Size "44"}
TYPE EL3164_B71BFF42 EXTENDS TcoIo.EtcSlaveTerminalBase_947E5A46 :
STRUCT
    {attribute addProperty Name "AI_Standard_Channel_1"}
    AI_Standard_Channel_1 : AI_Standard_Channel_A8DF64E3;
    {attribute addProperty Name "AI_Standard_Channel_2"}
    AI_Standard_Channel_2 : AI_Standard_Channel_A8DF64E3;
    {attribute addProperty Name "AI_Standard_Channel_3"}
    AI_Standard_Channel_3 : AI_Standard_Channel_A8DF64E3;
    {attribute addProperty Name "AI_Standard_Channel_4"}
    AI_Standard_Channel_4 : AI_Standard_Channel_A8DF64E3;
    {attribute addProperty Name "WcState"}
    WcState : TcoIo.WcState_9091E0EB;
    {attribute addProperty Name "InfoData"}
    InfoData : TcoIo.InfoData_23CBA837;
END_STRUCT
END_TYPE

// ---- DUTs/IO/Boxes/EL3403_812980A6.TcDUT
{attribute 'GeneratedUsingTerminal: EL3403-0000-0023'}
{attribute addProperty VendorId "#x00000002"}
{attribute addProperty BoxType "EL3403-0000-0023"}
{attribute addProperty Description "EL3403 3Ch. Power Measuring"}
{attribute addProperty Physics "KK"}
{attribute addProperty Id "PM_Inputs_Channel_1AT %I*PM_Inputs_Channel_2F86808618PM_Inputs_Channel_2AT %I*PM_Inputs_Channel_2F86808618PM_Inputs_Channel_3AT %I*PM_Inputs_Channel_2F86808618PM_Status_dataAT %I*PM_Status_data_2A9514CB4PM_Outputs_Channel_1AT %Q*PM_Outputs_Channel_E5FBDE301PM_Outputs_Channel_2AT %Q*PM_Outputs_Channel_E5FBDE301PM_Outputs_Channel_3AT %Q*PM_Outputs_Channel_E5FBDE301WcStateAT %I*WcState_9091E0EB2InfoDataAT %I*InfoData_23CBA8372"}
{attribute addProperty CRC "2166980774"}
{attribute addProperty Size "65"}
TYPE EL3403_812980A6 EXTENDS TcoIo.EtcSlaveTerminalBase_947E5A46 :
STRUCT
    {attribute addProperty Name "PM_Inputs_Channel_1"}
    PM_Inputs_Channel_1 : PM_Inputs_Channel_2F868086;
    {attribute addProperty Name "PM_Inputs_Channel_2"}
    PM_Inputs_Channel_2 : PM_Inputs_Channel_2F868086;
    {attribute addProperty Name "PM_Inputs_Channel_3"}
    PM_Inputs_Channel_3 : PM_Inputs_Channel_2F868086;
    {attribute addProperty Name "PM_Status_data"}
    PM_Status_data : PM_Status_data_2A9514CB;
    {attribute addProperty Name "PM_Outputs_Channel_1"}
    PM_Outputs_Channel_1 : PM_Outputs_Channel_E5FBDE30;
    {attribute addProperty Name "PM_Outputs_Channel_2"}
    PM_Outputs_Channel_2 : PM_Outputs_Channel_E5FBDE30;
    {attribute addProperty Name "PM_Outputs_Channel_3"}
    PM_Outputs_Channel_3 : PM_Outputs_Channel_E5FBDE30;
    {attribute addProperty Name "WcState"}
    WcState : TcoIo.WcState_9091E0EB;
    {attribute addProperty Name "InfoData"}
    InfoData : TcoIo.InfoData_23CBA837;
END_STRUCT
END_TYPE

// ---- DUTs/IO/Boxes/EL3024_C6E76B5A.TcDUT
{attribute 'GeneratedUsingTerminal: EL3024-0000-0018'}
{attribute addProperty VendorId "#x00000002"}
{attribute addProperty BoxType "EL3024-0000-0018"}
{attribute addProperty Description "EL3024 4Ch. Ana. Input 4-20mA DIFF"}
{attribute addProperty Physics "KK"}
{attribute addProperty Id "AI_Standard_Channel_1AT %I*AI_Standard_Channel_4A3944819AI_Standard_Channel_2AT %I*AI_Standard_Channel_4A3944819AI_Standard_Channel_3AT %I*AI_Standard_Channel_4A3944819AI_Standard_Channel_4AT %I*AI_Standard_Channel_4A3944819WcStateAT %I*WcState_9091E0EB2InfoDataAT %I*InfoData_23CBA8372"}
{attribute addProperty CRC "3337055066"}
{attribute addProperty Size "40"}
TYPE EL3024_C6E76B5A EXTENDS TcoIo.EtcSlaveTerminalBase_947E5A46 :
STRUCT
    {attribute addProperty Name "AI_Standard_Channel_1"}
    AI_Standard_Channel_1 : AI_Standard_Channel_4A394481;
    {attribute addProperty Name "AI_Standard_Channel_2"}
    AI_Standard_Channel_2 : AI_Standard_Channel_4A394481;
    {attribute addProperty Name "AI_Standard_Channel_3"}
    AI_Standard_Channel_3 : AI_Standard_Channel_4A394481;
    {attribute addProperty Name "AI_Standard_Channel_4"}
    AI_Standard_Channel_4 : AI_Standard_Channel_4A394481;
    {attribute addProperty Name "WcState"}
    WcState : TcoIo.WcState_9091E0EB;
    {attribute addProperty Name "InfoData"}
    InfoData : TcoIo.InfoData_23CBA837;
END_STRUCT
END_TYPE

// ---- DUTs/IO/Boxes/AX5101_1BD22F51.TcDUT
{attribute 'GeneratedUsingTerminal: AX5101-0000-0214-0214'}
{attribute addProperty VendorId "#x00000002"}
{attribute addProperty BoxType "AX5101-0000-0214-0214"}
{attribute addProperty Description "AX5101-0000-0214 EtherCAT Drive (SoE, 1 Ch.)"}
{attribute addProperty Physics "YY_K"}
{attribute addProperty Id "AT_xAT %I*AT_x_4EC2E76810MDTAT %Q*MDT_864618EC6WcStateAT %I*WcState_9091E0EB2InfoDataAT %I*InfoData_F60A43AC11"}
{attribute addProperty CRC "466759505"}
{attribute addProperty Size "29"}
TYPE AX5101_1BD22F51 EXTENDS TcoIo.EtcSlaveBoxBase_77A0E4A7 :
STRUCT
    {attribute addProperty Name "AT_x"}
    AT_x : AT_x_4EC2E768;
    {attribute addProperty Name "MDT"}
    MDT : MDT_864618EC;
    {attribute addProperty Name "WcState"}
    WcState : TcoIo.WcState_9091E0EB;
    {attribute addProperty Name "InfoData"}
    InfoData : InfoData_F60A43AC;
END_STRUCT
END_TYPE

// ---- DUTs/IO/Boxes/AX5106_1BD22F51.TcDUT
{attribute 'GeneratedUsingTerminal: AX5106-0000-0203-0203'}
{attribute addProperty VendorId "#x00000002"}
{attribute addProperty BoxType "AX5106-0000-0203-0203"}
{attribute addProperty Description "AX5106-0000-0203 EtherCAT Drive (SoE, 1 Ch.)"}
{attribute addProperty Physics "YY_K"}
{attribute addProperty Id "AT_xAT %I*AT_x_4EC2E76810MDTAT %Q*MDT_864618EC6WcStateAT %I*WcState_9091E0EB2InfoDataAT %I*InfoData_F60A43AC11"}
{attribute addProperty CRC "466759505"}
{attribute addProperty Size "29"}
TYPE AX5106_1BD22F51 EXTENDS TcoIo.EtcSlaveBoxBase_77A0E4A7 :
STRUCT
    {attribute addProperty Name "AT_x"}
    AT_x : AT_x_4EC2E768;
    {attribute addProperty Name "MDT"}
    MDT : MDT_864618EC;
    {attribute addProperty Name "WcState"}
    WcState : TcoIo.WcState_9091E0EB;
    {attribute addProperty Name "InfoData"}
    InfoData : InfoData_F60A43AC;
END_STRUCT
END_TYPE

// ---- DUTs/IO/Boxes/AES_A3B07071.TcDUT
{attribute 'GeneratedUsingTerminal: AES-D-BC-ECAT-0000'}
{attribute addProperty VendorId "#x00000024"}
{attribute addProperty BoxType "AES-D-BC-ECAT-0000"}
{attribute addProperty Description "AES Fieldbus Coupler"}
{attribute addProperty Physics "YY"}
{attribute addProperty Id "Module_1_32_Byte_Valve_Unit_0x7FModule_1_32_Byte_Valve_Unit_0x7F_1A3DA03C56Device_StateAT %I*Device_State_B9CC77574Device_ControlAT %Q*Device_Control_33EFE70E4WcStateAT %I*WcState_9091E0EB2InfoDataAT %I*InfoData_23CBA8372"}
{attribute addProperty CRC "2746249329"}
{attribute addProperty Size "68"}
TYPE AES_A3B07071 EXTENDS TcoIo.EtcSlaveBoxBase_77A0E4A7 :
STRUCT
    {attribute addProperty Name "Module_1_32_Byte_Valve_Unit_0x7F"}
    Module_1_32_Byte_Valve_Unit_0x7F : Module_1_32_Byte_Valve_Unit_0x7F_1A3DA03C;
    {attribute addProperty Name "Device_State"}
    Device_State : Device_State_B9CC7757;
    {attribute addProperty Name "Device_Control"}
    Device_Control : Device_Control_33EFE70E;
    {attribute addProperty Name "WcState"}
    WcState : TcoIo.WcState_9091E0EB;
    {attribute addProperty Name "InfoData"}
    InfoData : TcoIo.InfoData_23CBA837;
END_STRUCT
END_TYPE

// ---- DUTs/IO/Boxes/EL6631_A0EC075C.TcDUT
{attribute 'GeneratedUsingTerminal: EL6631-0000-0018'}
{attribute addProperty VendorId "#x00000002"}
{attribute addProperty BoxType "EL6631-0000-0018"}
{attribute addProperty Description "EL6631 PROFINET IO Controller"}
{attribute addProperty Physics "KK"}
{attribute addProperty Id "InfoDataAT %I*InfoData_8F85596B2"}
{attribute addProperty CRC "2699822940"}
{attribute addProperty Size "2"}
TYPE EL6631_A0EC075C EXTENDS TcoIo.EtcSlaveTerminalBase_947E5A46 :
STRUCT
    {attribute addProperty Name "InfoData"}
    InfoData : InfoData_8F85596B;
END_STRUCT
END_TYPE

// ---- DUTs/IO/Boxes/EL9010_D29C2085.TcDUT
{attribute 'GeneratedUsingTerminal: EL9010--0000'}
{attribute addProperty VendorId "#x00000002"}
{attribute addProperty BoxType "EL9010--0000"}
{attribute addProperty Description "EL9010 End Terminal"}
{attribute addProperty Physics "K"}
{attribute addProperty Id "EL9010"}
{attribute addProperty CRC "3533447301"}
{attribute addProperty Size "0"}
TYPE EL9010_D29C2085 EXTENDS TcoIo.EtcSlaveEndTerminalBase_866C7F0C :
STRUCT
END_STRUCT
END_TYPE

// ---- DUTs/IO/Boxes/AES_B47A2610.TcDUT
{attribute 'GeneratedUsingTerminal: AES-D-BC-ECAT-0000'}
{attribute addProperty VendorId "#x00000024"}
{attribute addProperty BoxType "AES-D-BC-ECAT-0000"}
{attribute addProperty Description "AES Fieldbus Coupler"}
{attribute addProperty Physics "YY"}
{attribute addProperty Id "Module_1_32_Byte_Valve_Unit_0x7FModule_1_32_Byte_Valve_Unit_0x7F_85784B2764Device_StateAT %I*Device_State_384275F89Device_ControlAT %Q*Device_Control_5857DF0F3WcStateAT %I*WcState_9091E0EB2InfoDataAT %I*InfoData_23CBA8372"}
{attribute addProperty CRC "3027904016"}
{attribute addProperty Size "80"}
TYPE AES_B47A2610 EXTENDS TcoIo.EtcSlaveBoxBase_77A0E4A7 :
STRUCT
    {attribute addProperty Name "Module_1_32_Byte_Valve_Unit_0x7F"}
    Module_1_32_Byte_Valve_Unit_0x7F : Module_1_32_Byte_Valve_Unit_0x7F_85784B27;
    {attribute addProperty Name "Device_State"}
    Device_State : Device_State_384275F8;
    {attribute addProperty Name "Device_Control"}
    Device_Control : Device_Control_5857DF0F;
    {attribute addProperty Name "WcState"}
    WcState : TcoIo.WcState_9091E0EB;
    {attribute addProperty Name "InfoData"}
    InfoData : TcoIo.InfoData_23CBA837;
END_STRUCT
END_TYPE

// ---- DUTs/IO/Boxes/IMecat_x_75C6CB6B.TcDUT
{attribute 'GeneratedUsingTerminal: IMecat-0007-0001'}
{attribute addProperty VendorId "#x00000024"}
{attribute addProperty BoxType "IMecat-0007-0001"}
{attribute addProperty Description "IMecat"}
{attribute addProperty Physics "YY"}
{attribute addProperty Id "DI_TxPDO_MapAT %I*DI_TxPDO_Map_DF955083132DO_RxPDO_MapAT %Q*DO_RxPDO_Map_8BCFF4C934WcStateAT %I*WcState_9091E0EB2InfoDataAT %I*InfoData_23CBA8372"}
{attribute addProperty CRC "1975962475"}
{attribute addProperty Size "170"}
TYPE IMecat_x_75C6CB6B EXTENDS TcoIo.EtcSlaveBoxBase_77A0E4A7 :
STRUCT
    {attribute addProperty Name "DI_TxPDO_Map"}
    DI_TxPDO_Map : DI_TxPDO_Map_DF955083;
    {attribute addProperty Name "DO_RxPDO_Map"}
    DO_RxPDO_Map : DO_RxPDO_Map_8BCFF4C9;
    {attribute addProperty Name "WcState"}
    WcState : TcoIo.WcState_9091E0EB;
    {attribute addProperty Name "InfoData"}
    InfoData : TcoIo.InfoData_23CBA837;
END_STRUCT
END_TYPE

// ---- DUTs/IO/Boxes/AX5103_1BD22F51.TcDUT
{attribute 'GeneratedUsingTerminal: AX5103-0000-0203-0203'}
{attribute addProperty VendorId "#x00000002"}
{attribute addProperty BoxType "AX5103-0000-0203-0203"}
{attribute addProperty Description "AX5103-0000-0203 EtherCAT Drive (SoE, 1 Ch.)"}
{attribute addProperty Physics "YY_K"}
{attribute addProperty Id "AT_xAT %I*AT_x_4EC2E76810MDTAT %Q*MDT_864618EC6WcStateAT %I*WcState_9091E0EB2InfoDataAT %I*InfoData_F60A43AC11"}
{attribute addProperty CRC "466759505"}
{attribute addProperty Size "29"}
TYPE AX5103_1BD22F51 EXTENDS TcoIo.EtcSlaveBoxBase_77A0E4A7 :
STRUCT
    {attribute addProperty Name "AT_x"}
    AT_x : AT_x_4EC2E768;
    {attribute addProperty Name "MDT"}
    MDT : MDT_864618EC;
    {attribute addProperty Name "WcState"}
    WcState : TcoIo.WcState_9091E0EB;
    {attribute addProperty Name "InfoData"}
    InfoData : InfoData_F60A43AC;
END_STRUCT
END_TYPE

// ---- DUTs/IO/Boxes/EL7332_DFB2BED7.TcDUT
{attribute 'GeneratedUsingTerminal: EL7332-0000-0024'}
{attribute addProperty VendorId "#x00000002"}
{attribute addProperty BoxType "EL7332-0000-0024"}
{attribute addProperty Description "EL7332 2Ch. DC motor output stage (24V, 1.5A)"}
{attribute addProperty Physics "KK"}
{attribute addProperty Id "DCM_Status_Channel_1AT %I*DCM_Status_Channel_36ED096F11DCM_Synchron_info_data_Channel_1AT %I*DCM_Synchron_info_data_Channel_6FB37C884DCM_Status_Channel_2AT %I*DCM_Status_Channel_36ED096F11DCM_Synchron_info_data_Channel_2AT %I*DCM_Synchron_info_data_Channel_6FB37C884DCM_Control_Channel_1AT %Q*DCM_Control_Channel_5A8B50163DCM_Velocity_Channel_1AT %Q*DCM_Velocity_Channel_A47A3F412DCM_Control_Channel_2AT %Q*DCM_Control_Channel_5A8B50163DCM_Velocity_Channel_2AT %Q*DCM_Velocity_Channel_A47A3F412WcStateAT %I*WcState_9091E0EB2InfoDataAT %I*InfoData_F38373C94"}
{attribute addProperty CRC "3753033431"}
{attribute addProperty Size "46"}
TYPE EL7332_DFB2BED7 EXTENDS TcoIo.EtcSlaveTerminalBase_947E5A46 :
STRUCT
    {attribute addProperty Name "DCM_Status_Channel_1"}
    DCM_Status_Channel_1 : DCM_Status_Channel_36ED096F;
    {attribute addProperty Name "DCM_Synchron_info_data_Channel_1"}
    DCM_Synchron_info_data_Channel_1 : DCM_Synchron_info_data_Channel_6FB37C88;
    {attribute addProperty Name "DCM_Status_Channel_2"}
    DCM_Status_Channel_2 : DCM_Status_Channel_36ED096F;
    {attribute addProperty Name "DCM_Synchron_info_data_Channel_2"}
    DCM_Synchron_info_data_Channel_2 : DCM_Synchron_info_data_Channel_6FB37C88;
    {attribute addProperty Name "DCM_Control_Channel_1"}
    DCM_Control_Channel_1 : DCM_Control_Channel_5A8B5016;
    {attribute addProperty Name "DCM_Velocity_Channel_1"}
    DCM_Velocity_Channel_1 : DCM_Velocity_Channel_A47A3F41;
    {attribute addProperty Name "DCM_Control_Channel_2"}
    DCM_Control_Channel_2 : DCM_Control_Channel_5A8B5016;
    {attribute addProperty Name "DCM_Velocity_Channel_2"}
    DCM_Velocity_Channel_2 : DCM_Velocity_Channel_A47A3F41;
    {attribute addProperty Name "WcState"}
    WcState : TcoIo.WcState_9091E0EB;
    {attribute addProperty Name "InfoData"}
    InfoData : InfoData_F38373C9;
END_STRUCT
END_TYPE

// ---- DUTs/IO/Boxes/CMMP_93B92D52.TcDUT
{attribute 'GeneratedUsingTerminal: CMMP-AS V4p0 CiA402-0002'}
{attribute addProperty VendorId "#x0000001d"}
{attribute addProperty BoxType "CMMP-AS V4p0 CiA402-0002"}
{attribute addProperty Description "CMMP-AS V4p0 CiA402"}
{attribute addProperty Physics "YY"}
{attribute addProperty Id "InputsAT %I*Inputs_424E3ECB8Inputs_1AT %I*Inputs_845131828OutputsAT %Q*Outputs_3179CEF48WcStateAT %I*WcState_9091E0EB2InfoDataAT %I*InfoData_F60A43AC11"}
{attribute addProperty CRC "2478386514"}
{attribute addProperty Size "37"}
TYPE CMMP_93B92D52 EXTENDS TcoIo.EtcSlaveBoxBase_77A0E4A7 :
STRUCT
    {attribute addProperty Name "Inputs"}
    Inputs : Inputs_424E3ECB;
    {attribute addProperty Name "Inputs_1"}
    Inputs_1 : Inputs_84513182;
    {attribute addProperty Name "Outputs"}
    Outputs : Outputs_3179CEF4;
    {attribute addProperty Name "WcState"}
    WcState : TcoIo.WcState_9091E0EB;
    {attribute addProperty Name "InfoData"}
    InfoData : InfoData_F60A43AC;
END_STRUCT
END_TYPE

// ---- DUTs/IO/Boxes/Flexi_Gateway_GETC1_429ECB70.TcDUT
{attribute 'GeneratedUsingTerminal: Flexi Gateway GETC1-0001-0000'}
{attribute addProperty VendorId "#x01000056"}
{attribute addProperty BoxType "Flexi Gateway GETC1-0001-0000"}
{attribute addProperty Description "FLX0-GETC100"}
{attribute addProperty Physics "YY"}
{attribute addProperty Id "NewMessageFlagAT %I*NewMessageFlag_557A079F1Gateway_to_EtherCAT_Data_100_BytesAT %I*Gateway_to_EtherCAT_Data_100_Bytes_AE1F4D6F0EtherCAT_to_Gateway_Data_100_BytesAT %Q*EtherCAT_to_Gateway_Data_100_Bytes_44CA1D220WcStateAT %I*WcState_9091E0EB2InfoDataAT %I*InfoData_23CBA8372"}
{attribute addProperty CRC "1117703024"}
{attribute addProperty Size "5"}
TYPE Flexi_Gateway_GETC1_429ECB70 EXTENDS TcoIo.EtcSlaveBoxBase_77A0E4A7 :
STRUCT
    {attribute addProperty Name "NewMessageFlag"}
    NewMessageFlag : NewMessageFlag_557A079F;
    {attribute addProperty Name "Gateway_to_EtherCAT_Data_100_Bytes"}
    Gateway_to_EtherCAT_Data_100_Bytes : Gateway_to_EtherCAT_Data_100_Bytes_AE1F4D6F;
    {attribute addProperty Name "EtherCAT_to_Gateway_Data_100_Bytes"}
    EtherCAT_to_Gateway_Data_100_Bytes : EtherCAT_to_Gateway_Data_100_Bytes_44CA1D22;
    {attribute addProperty Name "WcState"}
    WcState : TcoIo.WcState_9091E0EB;
    {attribute addProperty Name "InfoData"}
    InfoData : TcoIo.InfoData_23CBA837;
END_STRUCT
END_TYPE

// ---- DUTs/IO/Boxes/EL7211_008D5C9A.TcDUT
{attribute 'GeneratedUsingTerminal: EL7211-0010-0032'}
{attribute addProperty VendorId "#x00000002"}
{attribute addProperty BoxType "EL7211-0010-0032"}
{attribute addProperty Description "EL7211-0010 1Ch. MDP742 Servo motor output stage with OCT (50V, 4.5A RMS)"}
{attribute addProperty Physics "KK"}
{attribute addProperty Id "FB_PositionAT %I*FB_Position_3FA094ED4DRV_StatuswordAT %I*DRV_Statusword_9B36FDFC2DRV_Following_error_actual_valueAT %I*DRV_Following_error_actual_value_5AA320BF4DRV_ControlwordAT %Q*DRV_Controlword_F3F147212DRV_Target_positionAT %Q*DRV_Target_position_05240F144WcStateAT %I*WcState_9091E0EB2InfoDataAT %I*InfoData_433F077712"}
{attribute addProperty CRC "9264282"}
{attribute addProperty Size "30"}
TYPE EL7211_008D5C9A EXTENDS TcoIo.EtcSlaveTerminalBase_947E5A46 :
STRUCT
    {attribute addProperty Name "FB_Position"}
    FB_Position : FB_Position_3FA094ED;
    {attribute addProperty Name "DRV_Statusword"}
    DRV_Statusword : DRV_Statusword_9B36FDFC;
    {attribute addProperty Name "DRV_Following_error_actual_value"}
    DRV_Following_error_actual_value : DRV_Following_error_actual_value_5AA320BF;
    {attribute addProperty Name "DRV_Controlword"}
    DRV_Controlword : DRV_Controlword_F3F14721;
    {attribute addProperty Name "DRV_Target_position"}
    DRV_Target_position : DRV_Target_position_05240F14;
    {attribute addProperty Name "WcState"}
    WcState : TcoIo.WcState_9091E0EB;
    {attribute addProperty Name "InfoData"}
    InfoData : InfoData_433F0777;
END_STRUCT
END_TYPE

// ---- DUTs/IO/Boxes/EL3692_73B94100.TcDUT
{attribute 'GeneratedUsingTerminal: EL3692-0000-0020'}
{attribute addProperty VendorId "#x00000002"}
{attribute addProperty BoxType "EL3692-0000-0020"}
{attribute addProperty Description "EL3692 2Ch. resistance measurement terminal"}
{attribute addProperty Physics "KK"}
{attribute addProperty Id "SAI_Inputs_Channel_1AT %I*SAI_Inputs_Channel_9DCD655714SAI_Range_Channel_1AT %I*SAI_Range_Channel_BDBF6DA92SAI_Inputs_Real_Channel_1AT %I*SAI_Inputs_Real_Channel_CCECF13D4SAI_Inputs_Channel_2AT %I*SAI_Inputs_Channel_9DCD655714SAI_Range_Channel_2AT %I*SAI_Range_Channel_BDBF6DA92SAI_Inputs_Real_Channel_2AT %I*SAI_Inputs_Real_Channel_CCECF13D4SAI_Range_Control_Channel_1AT %Q*SAI_Range_Control_Channel_F5D9BC224SAI_Range_Control_Channel_2AT %Q*SAI_Range_Control_Channel_F5D9BC224WcStateAT %I*WcState_9091E0EB2InfoDataAT %I*InfoData_23CBA8372"}
{attribute addProperty CRC "1941520640"}
{attribute addProperty Size "52"}
TYPE EL3692_73B94100 EXTENDS TcoIo.EtcSlaveTerminalBase_947E5A46 :
STRUCT
    {attribute addProperty Name "SAI_Inputs_Channel_1"}
    SAI_Inputs_Channel_1 : SAI_Inputs_Channel_9DCD6557;
    {attribute addProperty Name "SAI_Range_Channel_1"}
    SAI_Range_Channel_1 : SAI_Range_Channel_BDBF6DA9;
    {attribute addProperty Name "SAI_Inputs_Real_Channel_1"}
    SAI_Inputs_Real_Channel_1 : SAI_Inputs_Real_Channel_CCECF13D;
    {attribute addProperty Name "SAI_Inputs_Channel_2"}
    SAI_Inputs_Channel_2 : SAI_Inputs_Channel_9DCD6557;
    {attribute addProperty Name "SAI_Range_Channel_2"}
    SAI_Range_Channel_2 : SAI_Range_Channel_BDBF6DA9;
    {attribute addProperty Name "SAI_Inputs_Real_Channel_2"}
    SAI_Inputs_Real_Channel_2 : SAI_Inputs_Real_Channel_CCECF13D;
    {attribute addProperty Name "SAI_Range_Control_Channel_1"}
    SAI_Range_Control_Channel_1 : SAI_Range_Control_Channel_F5D9BC22;
    {attribute addProperty Name "SAI_Range_Control_Channel_2"}
    SAI_Range_Control_Channel_2 : SAI_Range_Control_Channel_F5D9BC22;
    {attribute addProperty Name "WcState"}
    WcState : TcoIo.WcState_9091E0EB;
    {attribute addProperty Name "InfoData"}
    InfoData : TcoIo.InfoData_23CBA837;
END_STRUCT
END_TYPE

// ---- DUTs/IO/Boxes/EPP1322_1FC0878B.TcDUT
{attribute 'GeneratedUsingTerminal: EPP1322-0001-0017'}
{attribute addProperty VendorId "#x00000002"}
{attribute addProperty BoxType "EPP1322-0001-0017"}
{attribute addProperty Description "EPP1322-0001 3 port EtherCAT P gateway"}
{attribute addProperty Physics "YYYY"}
{attribute addProperty Id "InfoDataAT %I*InfoData_6F19DB2B2"}
{attribute addProperty CRC "532711307"}
{attribute addProperty Size "2"}
TYPE EPP1322_1FC0878B EXTENDS TcoIo.EtcSlaveBoxBase_77A0E4A7 :
STRUCT
    {attribute addProperty Name "InfoData"}
    InfoData : TcoIo.InfoData_6F19DB2B;
END_STRUCT
END_TYPE

// ---- DUTs/IO/Boxes/EPP1008_78E8D3DD.TcDUT
{attribute 'GeneratedUsingTerminal: EPP1008-0001-0017'}
{attribute addProperty VendorId "#x00000002"}
{attribute addProperty BoxType "EPP1008-0001-0017"}
{attribute addProperty Description "EPP1008-0001 8 Ch. Dig. Input 24V, 3ms, M8"}
{attribute addProperty Physics "YY"}
{attribute addProperty Id "Channel_1AT %I*Channel_830843C11Channel_2AT %I*Channel_830843C11Channel_3AT %I*Channel_830843C11Channel_4AT %I*Channel_830843C11Channel_5AT %I*Channel_830843C11Channel_6AT %I*Channel_830843C11Channel_7AT %I*Channel_830843C11Channel_8AT %I*Channel_830843C11WcStateAT %I*WcState_9091E0EB2InfoDataAT %I*InfoData_6F19DB2B2"}
{attribute addProperty CRC "2028524509"}
{attribute addProperty Size "12"}
TYPE EPP1008_78E8D3DD EXTENDS TcoIo.EtcSlaveBoxBase_77A0E4A7 :
STRUCT
    {attribute addProperty Name "Channel_1"}
    Channel_1 : Channel_830843C1;
    {attribute addProperty Name "Channel_2"}
    Channel_2 : Channel_830843C1;
    {attribute addProperty Name "Channel_3"}
    Channel_3 : Channel_830843C1;
    {attribute addProperty Name "Channel_4"}
    Channel_4 : Channel_830843C1;
    {attribute addProperty Name "Channel_5"}
    Channel_5 : Channel_830843C1;
    {attribute addProperty Name "Channel_6"}
    Channel_6 : Channel_830843C1;
    {attribute addProperty Name "Channel_7"}
    Channel_7 : Channel_830843C1;
    {attribute addProperty Name "Channel_8"}
    Channel_8 : Channel_830843C1;
    {attribute addProperty Name "WcState"}
    WcState : TcoIo.WcState_9091E0EB;
    {attribute addProperty Name "InfoData"}
    InfoData : TcoIo.InfoData_6F19DB2B;
END_STRUCT
END_TYPE

// ---- DUTs/IO/Boxes/EPP1332_1FC0878B.TcDUT
{attribute 'GeneratedUsingTerminal: EPP1332-0001-0017'}
{attribute addProperty VendorId "#x00000002"}
{attribute addProperty BoxType "EPP1332-0001-0017"}
{attribute addProperty Description "EPP1332-0001 3 port EtherCAT P junction, power refreshing"}
{attribute addProperty Physics "YYYY"}
{attribute addProperty Id "InfoDataAT %I*InfoData_6F19DB2B2"}
{attribute addProperty CRC "532711307"}
{attribute addProperty Size "2"}
TYPE EPP1332_1FC0878B EXTENDS TcoIo.EtcSlaveBoxBase_77A0E4A7 :
STRUCT
    {attribute addProperty Name "InfoData"}
    InfoData : TcoIo.InfoData_6F19DB2B;
END_STRUCT
END_TYPE

// ---- DUTs/IO/Boxes/Flexi_Soft_EtherCAT_Gateway_DE394EDD.TcDUT
{attribute 'GeneratedUsingTerminal: Flexi Soft EtherCAT Gateway-0000-0001'}
{attribute addProperty VendorId "#x01000056"}
{attribute addProperty BoxType "Flexi Soft EtherCAT Gateway-0000-0001"}
{attribute addProperty Description "Flexi Soft EtherCAT Gateway"}
{attribute addProperty Physics "YY"}
{attribute addProperty Id "InAT %I*In_389F2F151OutAT %Q*Out_81AAEF2D0WcStateAT %I*WcState_9091E0EB2InfoDataAT %I*InfoData_23CBA8372"}
{attribute addProperty CRC "3728297693"}
{attribute addProperty Size "5"}
TYPE Flexi_Soft_EtherCAT_Gateway_DE394EDD EXTENDS TcoIo.EtcSlaveBoxBase_77A0E4A7 :
STRUCT
    {attribute addProperty Name "In"}
    In : In_389F2F15;
    {attribute addProperty Name "Out"}
    Out : Out_81AAEF2D;
    {attribute addProperty Name "WcState"}
    WcState : TcoIo.WcState_9091E0EB;
    {attribute addProperty Name "InfoData"}
    InfoData : TcoIo.InfoData_23CBA837;
END_STRUCT
END_TYPE

// ---- DUTs/IO/Boxes/EL7041_86DE63E7.TcDUT
{attribute 'GeneratedUsingTerminal: EL7041-1000-0021'}
{attribute addProperty VendorId "#x00000002"}
{attribute addProperty BoxType "EL7041-1000-0021"}
{attribute addProperty Description "EL7041-1000 1Ch. Stepper motor output stage (50V, 5A, standard)"}
{attribute addProperty Physics "KK"}
{attribute addProperty Id "ENC_Status_compactAT %I*ENC_Status_compact_4D066E1A16STM_StatusAT %I*STM_Status_36ED096F11ENC_Control_compactAT %Q*ENC_Control_compact_21E2D14D6STM_ControlAT %Q*STM_Control_5A8B50163STM_VelocityAT %Q*STM_Velocity_A47A3F412WcStateAT %I*WcState_9091E0EB2InfoDataAT %I*InfoData_D50C85453"}
{attribute addProperty CRC "2262721511"}
{attribute addProperty Size "43"}
TYPE EL7041_86DE63E7 EXTENDS TcoIo.EtcSlaveTerminalBase_947E5A46 :
STRUCT
    {attribute addProperty Name "ENC_Status_compact"}
    ENC_Status_compact : ENC_Status_compact_4D066E1A;
    {attribute addProperty Name "STM_Status"}
    STM_Status : STM_Status_36ED096F;
    {attribute addProperty Name "ENC_Control_compact"}
    ENC_Control_compact : ENC_Control_compact_21E2D14D;
    {attribute addProperty Name "STM_Control"}
    STM_Control : STM_Control_5A8B5016;
    {attribute addProperty Name "STM_Velocity"}
    STM_Velocity : STM_Velocity_A47A3F41;
    {attribute addProperty Name "WcState"}
    WcState : TcoIo.WcState_9091E0EB;
    {attribute addProperty Name "InfoData"}
    InfoData : InfoData_D50C8545;
END_STRUCT
END_TYPE

// ---- DUTs/IO/Boxes/IndraDrive_MPB20_C66205C3.TcDUT
{attribute 'GeneratedUsingTerminal: IndraDrive MPB20-0003-0000'}
{attribute addProperty VendorId "#x00000024"}
{attribute addProperty BoxType "IndraDrive MPB20-0003-0000"}
{attribute addProperty Description "IndraDrive MPB20"}
{attribute addProperty Physics "YY"}
{attribute addProperty Id "AT_xAT %I*AT_x_26CC547D6MDTAT %Q*MDT_864618EC6WcStateAT %I*WcState_9091E0EB2InfoDataAT %I*InfoData_F60A43AC11"}
{attribute addProperty CRC "3328312771"}
{attribute addProperty Size "25"}
TYPE IndraDrive_MPB20_C66205C3 EXTENDS TcoIo.EtcSlaveBoxBase_77A0E4A7 :
STRUCT
    {attribute addProperty Name "AT_x"}
    AT_x : AT_x_26CC547D;
    {attribute addProperty Name "MDT"}
    MDT : MDT_864618EC;
    {attribute addProperty Name "WcState"}
    WcState : TcoIo.WcState_9091E0EB;
    {attribute addProperty Name "InfoData"}
    InfoData : InfoData_F60A43AC;
END_STRUCT
END_TYPE

// ---- DUTs/IO/Boxes/EPP2308_F6D9A8D1.TcDUT
{attribute 'GeneratedUsingTerminal: EPP2308-0001-0018'}
{attribute addProperty VendorId "#x00000002"}
{attribute addProperty BoxType "EPP2308-0001-0018"}
{attribute addProperty Description "EPP2308-0001 4 Ch. Dig. In, 3ms, 4 Ch. Dig. Out 24V, 0,5A, M8"}
{attribute addProperty Physics "YY"}
{attribute addProperty Id "Channel_1AT %I*Channel_830843C11Channel_2AT %I*Channel_830843C11Channel_3AT %I*Channel_830843C11Channel_4AT %I*Channel_830843C11Channel_5AT %Q*Channel_42CA91F71Channel_6AT %Q*Channel_42CA91F71Channel_7AT %Q*Channel_42CA91F71Channel_8AT %Q*Channel_42CA91F71WcStateAT %I*WcState_9091E0EB2InfoDataAT %I*InfoData_6F19DB2B2"}
{attribute addProperty CRC "4141459665"}
{attribute addProperty Size "12"}
TYPE EPP2308_F6D9A8D1 EXTENDS TcoIo.EtcSlaveBoxBase_77A0E4A7 :
STRUCT
    {attribute addProperty Name "Channel_1"}
    Channel_1 : Channel_830843C1;
    {attribute addProperty Name "Channel_2"}
    Channel_2 : Channel_830843C1;
    {attribute addProperty Name "Channel_3"}
    Channel_3 : Channel_830843C1;
    {attribute addProperty Name "Channel_4"}
    Channel_4 : Channel_830843C1;
    {attribute addProperty Name "Channel_5"}
    Channel_5 : Channel_42CA91F7;
    {attribute addProperty Name "Channel_6"}
    Channel_6 : Channel_42CA91F7;
    {attribute addProperty Name "Channel_7"}
    Channel_7 : Channel_42CA91F7;
    {attribute addProperty Name "Channel_8"}
    Channel_8 : Channel_42CA91F7;
    {attribute addProperty Name "WcState"}
    WcState : TcoIo.WcState_9091E0EB;
    {attribute addProperty Name "InfoData"}
    InfoData : TcoIo.InfoData_6F19DB2B;
END_STRUCT
END_TYPE

// ---- DUTs/IO/Devices/SyncUnitTasks_5FDC9770.TcDUT
{attribute 'GeneratedUsingTerminal: '}
{attribute addProperty BoxType ""}
{attribute addProperty Id "unreferencedAT %I*SyncUnitTask_AB2F50799PlcTask1AT %I*SyncUnitTask_AB2F50799"}
{attribute addProperty CRC "1608292208"}
{attribute addProperty Size "18"}
TYPE SyncUnitTasks_5FDC9770 EXTENDS TcoIo.SyncUnitTasksBase_7C8711EB :
STRUCT
    {attribute addProperty Name "unreferenced"}
    unreferenced : TcoIo.SyncUnitTask_AB2F5079;
    {attribute addProperty Name "PlcTask1"}
    PlcTask1 : TcoIo.SyncUnitTask_AB2F5079;
END_STRUCT
END_TYPE

// ---- DUTs/IO/Devices/SyncUnits_C3A34B50.TcDUT
{attribute 'GeneratedUsingTerminal: '}
{attribute addProperty BoxType ""}
{attribute addProperty Id "_defaultAT %I*SyncUnitTasks_5FDC977018"}
{attribute addProperty CRC "3282258768"}
{attribute addProperty Size "18"}
TYPE SyncUnits_C3A34B50 EXTENDS TcoIo.SyncUnitsBase_AD6C35CE :
STRUCT
    {attribute addProperty Name "_default"}
    _default : SyncUnitTasks_5FDC9770;
END_STRUCT
END_TYPE

// ---- DUTs/IO/Devices/SyncUnits_F0D163CC.TcDUT
{attribute 'GeneratedUsingTerminal: '}
{attribute addProperty BoxType ""}
{attribute addProperty Id "_defaultAT %I*SyncUnitTasks_5FDC977018Row_0AT %I*SyncUnitTasks_5FDC977018Row_1AT %I*SyncUnitTasks_5FDC977018Row_2AT %I*SyncUnitTasks_5FDC977018Row_3AT %I*SyncUnitTasks_5FDC977018Row_4AT %I*SyncUnitTasks_5FDC977018"}
{attribute addProperty CRC "4040254412"}
{attribute addProperty Size "108"}
TYPE SyncUnits_F0D163CC EXTENDS TcoIo.SyncUnitsBase_AD6C35CE :
STRUCT
    {attribute addProperty Name "_default"}
    _default : SyncUnitTasks_5FDC9770;
    {attribute addProperty Name "Row_0"}
    Row_0 : SyncUnitTasks_5FDC9770;
    {attribute addProperty Name "Row_1"}
    Row_1 : SyncUnitTasks_5FDC9770;
    {attribute addProperty Name "Row_2"}
    Row_2 : SyncUnitTasks_5FDC9770;
    {attribute addProperty Name "Row_3"}
    Row_3 : SyncUnitTasks_5FDC9770;
    {attribute addProperty Name "Row_4"}
    Row_4 : SyncUnitTasks_5FDC9770;
END_STRUCT
END_TYPE

// ---- DUTs/IO/Devices/SyncUnits_5BE71B8B.TcDUT
{attribute 'GeneratedUsingTerminal: '}
{attribute addProperty BoxType ""}
{attribute addProperty Id "_defaultAT %I*SyncUnitTasks_5FDC977018N10AT %I*SyncUnitTasks_5FDC977018S10AT %I*SyncUnitTasks_5FDC977018P10AT %I*SyncUnitTasks_5FDC977018P20AT %I*SyncUnitTasks_5FDC977018P30AT %I*SyncUnitTasks_5FDC977018C10AT %I*SyncUnitTasks_5FDC977018C20AT %I*SyncUnitTasks_5FDC977018C30AT %I*SyncUnitTasks_5FDC977018C40AT %I*SyncUnitTasks_5FDC977018C50AT %I*SyncUnitTasks_5FDC977018C60AT %I*SyncUnitTasks_5FDC977018C70AT %I*SyncUnitTasks_5FDC977018C80AT %I*SyncUnitTasks_5FDC977018R10AT %I*SyncUnitTasks_5FDC977018RHAT %I*SyncUnitTasks_5FDC977018"}
{attribute addProperty CRC "1541872523"}
{attribute addProperty Size "288"}
TYPE SyncUnits_5BE71B8B EXTENDS TcoIo.SyncUnitsBase_AD6C35CE :
STRUCT
    {attribute addProperty Name "_default"}
    _default : SyncUnitTasks_5FDC9770;
    {attribute addProperty Name "N10"}
    N10 : SyncUnitTasks_5FDC9770;
    {attribute addProperty Name "S10"}
    S10 : SyncUnitTasks_5FDC9770;
    {attribute addProperty Name "P10"}
    P10 : SyncUnitTasks_5FDC9770;
    {attribute addProperty Name "P20"}
    P20 : SyncUnitTasks_5FDC9770;
    {attribute addProperty Name "P30"}
    P30 : SyncUnitTasks_5FDC9770;
    {attribute addProperty Name "C10"}
    C10 : SyncUnitTasks_5FDC9770;
    {attribute addProperty Name "C20"}
    C20 : SyncUnitTasks_5FDC9770;
    {attribute addProperty Name "C30"}
    C30 : SyncUnitTasks_5FDC9770;
    {attribute addProperty Name "C40"}
    C40 : SyncUnitTasks_5FDC9770;
    {attribute addProperty Name "C50"}
    C50 : SyncUnitTasks_5FDC9770;
    {attribute addProperty Name "C60"}
    C60 : SyncUnitTasks_5FDC9770;
    {attribute addProperty Name "C70"}
    C70 : SyncUnitTasks_5FDC9770;
    {attribute addProperty Name "C80"}
    C80 : SyncUnitTasks_5FDC9770;
    {attribute addProperty Name "R10"}
    R10 : SyncUnitTasks_5FDC9770;
    {attribute addProperty Name "RH"}
    RH : SyncUnitTasks_5FDC9770;
END_STRUCT
END_TYPE

// ---- DUTs/IO/Topology/Term_1_EK1200_B38DC9A8.TcDUT
{attribute 'GeneratedUsingTerminal: EK1200-1388-0000'}
{attribute addProperty BoxType "EK1200-1388-0000"}
{attribute addProperty Id "Term_2_EL6002EL6002_CD897635118Term_3_EL1809EL1809_32157CFD20Term_4_EL2809EL2809_2B6483BD19Term_5_EL4004EL4004_E203F87511Term_6_EL2809EL2809_2B6483BD19Term_7_EL6001EL6001_0DE01E7E61Term_8_EL9011EL9011_D65D3D320"}
{attribute addProperty CRC "3012413864"}
{attribute addProperty Size "248"}
{attribute addProperty Name "Term 1 (EK1200)"}
TYPE Term_1_EK1200_B38DC9A8 EXTENDS EK1200_013D0B49 :
STRUCT
    {attribute addProperty Name "Term 2 (EL6002)"}
    {attribute addProperty PreviousPort "Term 1 (EK1200) : B"}
    {attribute addProperty SyncUnit "default"}
    Term_2_EL6002 : EL6002_CD897635;
    {attribute addProperty Name "Term 3 (EL1809)"}
    {attribute addProperty PreviousPort "Term 2 (EL6002) : B"}
    {attribute addProperty SyncUnit "default"}
    Term_3_EL1809 : EL1809_32157CFD;
    {attribute addProperty Name "Term 4 (EL2809)"}
    {attribute addProperty PreviousPort "Term 3 (EL1809) : B"}
    {attribute addProperty SyncUnit "default"}
    Term_4_EL2809 : EL2809_2B6483BD;
    {attribute addProperty Name "Term 5 (EL4004)"}
    {attribute addProperty PreviousPort "Term 4 (EL2809) : B"}
    {attribute addProperty SyncUnit "default"}
    Term_5_EL4004 : EL4004_E203F875;
    {attribute addProperty Name "Term 6 (EL2809)"}
    {attribute addProperty PreviousPort "Term 5 (EL4004) : B"}
    {attribute addProperty SyncUnit "default"}
    Term_6_EL2809 : EL2809_2B6483BD;
    {attribute addProperty Name "Term 7 (EL6001)"}
    {attribute addProperty PreviousPort "Term 6 (EL2809) : B"}
    {attribute addProperty SyncUnit "default"}
    Term_7_EL6001 : EL6001_0DE01E7E;
    {attribute addProperty Name "Term 8 (EL9011)"}
    {attribute addProperty PreviousPort "Term 7 (EL6001) : B"}
    {attribute addProperty SyncUnit "default"}
    Term_8_EL9011 : EL9011_D65D3D32;
END_STRUCT
END_TYPE

// ---- DUTs/IO/Topology/Device_1_EtherCAT_49C09C66.TcDUT
{attribute 'GeneratedUsingTerminal: IODEVICETYPE_ETHERCATPROT'}
{attribute addProperty BoxType "IODEVICETYPE_ETHERCATPROT"}
{attribute addProperty Id "Term_1_EK1200Term_1_EK1200_B38DC9A8248SyncUnitsSyncUnits_C3A34B5018InputsInputs_A65FACA410OutputsOutputs_23C0ED1D6InfoDataInfoData_84133AC922"}
{attribute addProperty CRC "1237359718"}
{attribute addProperty Size "304"}
{attribute addProperty Name "Device 1 (EtherCAT)"}
TYPE Device_1_EtherCAT_49C09C66 EXTENDS TcoIo.EtcMasterBase_62654B43 :
STRUCT
    {attribute addProperty Name "Term 1 (EK1200)"}
    {attribute addProperty PreviousPort "Device 1 (EtherCAT) : Master"}
    {attribute addProperty SyncUnit "default"}
    Term_1_EK1200 : Term_1_EK1200_B38DC9A8;
    {attribute addProperty Name "SyncUnits"}
    SyncUnits : SyncUnits_C3A34B50;
    {attribute addProperty Name "Inputs"}
    Inputs : TcoIo.Inputs_A65FACA4;
    {attribute addProperty Name "Outputs"}
    Outputs : TcoIo.Outputs_23C0ED1D;
    {attribute addProperty Name "InfoData"}
    InfoData : TcoIo.InfoData_84133AC9;
END_STRUCT
END_TYPE

// ---- DUTs/IO/Topology/Term_11_EK1100_B6553301.TcDUT
{attribute 'GeneratedUsingTerminal: EK1100-0000-0018'}
{attribute addProperty BoxType "EK1100-0000-0018"}
{attribute addProperty Id "Term_12_EL3174_0002EL3174_B71BFF4244Term_13_EL6001EL6001_0DE01E7E61Term_14_EL3011EL3011_7A49522813Term_15_EL2008EL2008_E2806B9511Term_16_EL2008EL2008_E2806B9511Term_17_EK1110EK1110_1FC0878B2"}
{attribute addProperty CRC "3059036929"}
{attribute addProperty Size "142"}
{attribute addProperty Name "Term 11 (EK1100)"}
TYPE Term_11_EK1100_B6553301 EXTENDS EK1100_1FC0878B :
STRUCT
    {attribute addProperty Name "Term 12 (EL3174-0002)"}
    {attribute addProperty PreviousPort "Term 11 (EK1100) : B"}
    {attribute addProperty SyncUnit "Row_1"}
    Term_12_EL3174_0002 : EL3174_B71BFF42;
    {attribute addProperty Name "Term 13 (EL6001)"}
    {attribute addProperty PreviousPort "Term 12 (EL3174-0002) : B"}
    {attribute addProperty SyncUnit "Row_1"}
    Term_13_EL6001 : EL6001_0DE01E7E;
    {attribute addProperty Name "Term 14 (EL3011)"}
    {attribute addProperty PreviousPort "Term 13 (EL6001) : B"}
    {attribute addProperty SyncUnit "Row_1"}
    Term_14_EL3011 : EL3011_7A495228;
    {attribute addProperty Name "Term 15 (EL2008)"}
    {attribute addProperty PreviousPort "Term 14 (EL3011) : B"}
    {attribute addProperty SyncUnit "Row_1"}
    Term_15_EL2008 : EL2008_E2806B95;
    {attribute addProperty Name "Term 16 (EL2008)"}
    {attribute addProperty PreviousPort "Term 15 (EL2008) : B"}
    {attribute addProperty SyncUnit "Row_1"}
    Term_16_EL2008 : EL2008_E2806B95;
    {attribute addProperty Name "Term 17 (EK1110)"}
    {attribute addProperty PreviousPort "Term 16 (EL2008) : B"}
    {attribute addProperty SyncUnit "default"}
    Term_17_EK1110 : EK1110_1FC0878B;
END_STRUCT
END_TYPE

// ---- DUTs/IO/Topology/Term_18_EK1100_20659A8D.TcDUT
{attribute 'GeneratedUsingTerminal: EK1100-0000-0018'}
{attribute addProperty BoxType "EK1100-0000-0018"}
{attribute addProperty Id "Term_19_EL1809EL1809_32157CFD20Term_20_EL2809EL2809_2B6483BD19Term_21_EL1809EL1809_32157CFD20Term_22_EL3011EL3011_7A49522813Term_29_EL9011EL9011_D65D3D320"}
{attribute addProperty CRC "543529613"}
{attribute addProperty Size "72"}
{attribute addProperty Name "Term 18 (EK1100)"}
TYPE Term_18_EK1100_20659A8D EXTENDS EK1100_1FC0878B :
STRUCT
    {attribute addProperty Name "Term 19 (EL1809)"}
    {attribute addProperty PreviousPort "Term 18 (EK1100) : B"}
    {attribute addProperty SyncUnit "Row_1"}
    Term_19_EL1809 : EL1809_32157CFD;
    {attribute addProperty Name "Term 20 (EL2809)"}
    {attribute addProperty PreviousPort "Term 19 (EL1809) : B"}
    {attribute addProperty SyncUnit "Row_1"}
    Term_20_EL2809 : EL2809_2B6483BD;
    {attribute addProperty Name "Term 21 (EL1809)"}
    {attribute addProperty PreviousPort "Term 20 (EL2809) : B"}
    {attribute addProperty SyncUnit "Row_1"}
    Term_21_EL1809 : EL1809_32157CFD;
    {attribute addProperty Name "Term 22 (EL3011)"}
    {attribute addProperty PreviousPort "Term 21 (EL1809) : B"}
    {attribute addProperty SyncUnit "Row_1"}
    Term_22_EL3011 : EL3011_7A495228;
    {attribute addProperty Name "Term 29 (EL9011)"}
    {attribute addProperty PreviousPort "Term 22 (EL3011) : B"}
    {attribute addProperty SyncUnit "default"}
    Term_29_EL9011 : EL9011_D65D3D32;
END_STRUCT
END_TYPE

// ---- DUTs/IO/Topology/Term_25_EK1100_08217EB4.TcDUT
{attribute 'GeneratedUsingTerminal: EK1100-0000-0018'}
{attribute addProperty BoxType "EK1100-0000-0018"}
{attribute addProperty Id "Term_26_EL1819EL1819_32157CFD20Term_27_EL1819EL1819_32157CFD20Term_30_EL9011EL9011_D65D3D320"}
{attribute addProperty CRC "136412852"}
{attribute addProperty Size "40"}
{attribute addProperty Name "Term 25 (EK1100)"}
TYPE Term_25_EK1100_08217EB4 EXTENDS EK1100_1FC0878B :
STRUCT
    {attribute addProperty Name "Term 26 (EL1819)"}
    {attribute addProperty PreviousPort "Term 25 (EK1100) : B"}
    {attribute addProperty SyncUnit "Row_3"}
    Term_26_EL1819 : EL1819_32157CFD;
    {attribute addProperty Name "Term 27 (EL1819)"}
    {attribute addProperty PreviousPort "Term 26 (EL1819) : B"}
    {attribute addProperty SyncUnit "Row_3"}
    Term_27_EL1819 : EL1819_32157CFD;
    {attribute addProperty Name "Term 30 (EL9011)"}
    {attribute addProperty PreviousPort "Term 27 (EL1819) : B"}
    {attribute addProperty SyncUnit "default"}
    Term_30_EL9011 : EL9011_D65D3D32;
END_STRUCT
END_TYPE

// ---- DUTs/IO/Topology/Term_28_EK1100_415F4A7E.TcDUT
{attribute 'GeneratedUsingTerminal: EK1100-0000-0018'}
{attribute addProperty BoxType "EK1100-0000-0018"}
{attribute addProperty Id "Term_29_EL2788EL2788_E2806B9511Term_30_EL3773EL3773_F128CC82184Term_31_EL9011EL9011_D65D3D320"}
{attribute addProperty CRC "1096764030"}
{attribute addProperty Size "195"}
{attribute addProperty Name "Term 28 (EK1100)"}
TYPE Term_28_EK1100_415F4A7E EXTENDS EK1100_1FC0878B :
STRUCT
    {attribute addProperty Name "Term 29 (EL2788)"}
    {attribute addProperty PreviousPort "Term 28 (EK1100) : B"}
    {attribute addProperty SyncUnit "Row_4"}
    Term_29_EL2788 : EL2788_E2806B95;
    {attribute addProperty Name "Term 30 (EL3773)"}
    {attribute addProperty PreviousPort "Term 29 (EL2788) : B"}
    {attribute addProperty SyncUnit "Row_4"}
    Term_30_EL3773 : EL3773_F128CC82;
    {attribute addProperty Name "Term 31 (EL9011)"}
    {attribute addProperty PreviousPort "Term 30 (EL3773) : B"}
    {attribute addProperty SyncUnit "default"}
    Term_31_EL9011 : EL9011_D65D3D32;
END_STRUCT
END_TYPE

// ---- DUTs/IO/Topology/Term_24_EK1122_39E7B5CB.TcDUT
{attribute 'GeneratedUsingTerminal: EK1122-0000-0018'}
{attribute addProperty BoxType "EK1122-0000-0018"}
{attribute addProperty Id "Term_25_EK1100Term_25_EK1100_08217EB440Term_28_EK1100Term_28_EK1100_415F4A7E195"}
{attribute addProperty CRC "971486667"}
{attribute addProperty Size "235"}
{attribute addProperty Name "Term 24 (EK1122)"}
TYPE Term_24_EK1122_39E7B5CB EXTENDS EK1122_1FC0878B :
STRUCT
    {attribute addProperty Name "Term 25 (EK1100)"}
    {attribute addProperty PreviousPort "Term 24 (EK1122) : B"}
    {attribute addProperty SyncUnit "default"}
    Term_25_EK1100 : Term_25_EK1100_08217EB4;
    {attribute addProperty Name "Term 28 (EK1100)"}
    {attribute addProperty PreviousPort "Term 25 (EK1100) : C"}
    {attribute addProperty SyncUnit "default"}
    Term_28_EK1100 : Term_28_EK1100_415F4A7E;
END_STRUCT
END_TYPE

// ---- DUTs/IO/Topology/Term_23_EK1100_DFBF0BE4.TcDUT
{attribute 'GeneratedUsingTerminal: EK1100-0000-0018'}
{attribute addProperty BoxType "EK1100-0000-0018"}
{attribute addProperty Id "Term_24_EK1122Term_24_EK1122_39E7B5CB235Term_31_EL3773EL3773_F128CC82184Term_32_EL2258EL2258_E3B260FA508Term_33_EL3164EL3164_B71BFF4244Term_32_EL9011EL9011_D65D3D320"}
{attribute addProperty CRC "3753839588"}
{attribute addProperty Size "971"}
{attribute addProperty Name "Term 23 (EK1100)"}
TYPE Term_23_EK1100_DFBF0BE4 EXTENDS EK1100_1FC0878B :
STRUCT
    {attribute addProperty Name "Term 24 (EK1122)"}
    {attribute addProperty PreviousPort "Term 23 (EK1100) : B"}
    {attribute addProperty SyncUnit "default"}
    Term_24_EK1122 : Term_24_EK1122_39E7B5CB;
    {attribute addProperty Name "Term 31 (EL3773)"}
    {attribute addProperty PreviousPort "Term 24 (EK1122) : C"}
    {attribute addProperty SyncUnit "Row_2"}
    Term_31_EL3773 : EL3773_F128CC82;
    {attribute addProperty Name "Term 32 (EL2258)"}
    {attribute addProperty PreviousPort "Term 31 (EL3773) : B"}
    {attribute addProperty SyncUnit "Row_2"}
    Term_32_EL2258 : EL2258_E3B260FA;
    {attribute addProperty Name "Term 33 (EL3164)"}
    {attribute addProperty PreviousPort "Term 32 (EL2258) : B"}
    {attribute addProperty SyncUnit "Row_2"}
    Term_33_EL3164 : EL3164_B71BFF42;
    {attribute addProperty Name "Term 32 (EL9011)"}
    {attribute addProperty PreviousPort "Term 33 (EL3164) : B"}
    {attribute addProperty SyncUnit "default"}
    Term_32_EL9011 : EL9011_D65D3D32;
END_STRUCT
END_TYPE

// ---- DUTs/IO/Topology/Term_10_EK1122_3D069EC1.TcDUT
{attribute 'GeneratedUsingTerminal: EK1122-0000-0018'}
{attribute addProperty BoxType "EK1122-0000-0018"}
{attribute addProperty Id "Term_11_EK1100Term_11_EK1100_B6553301142Term_18_EK1100Term_18_EK1100_20659A8D72Term_23_EK1100Term_23_EK1100_DFBF0BE4971"}
{attribute addProperty CRC "1023844033"}
{attribute addProperty Size "1185"}
{attribute addProperty Name "Term 10 (EK1122)"}
TYPE Term_10_EK1122_3D069EC1 EXTENDS EK1122_1FC0878B :
STRUCT
    {attribute addProperty Name "Term 11 (EK1100)"}
    {attribute addProperty PreviousPort "Term 10 (EK1122) : D"}
    {attribute addProperty SyncUnit "default"}
    Term_11_EK1100 : Term_11_EK1100_B6553301;
    {attribute addProperty Name "Term 18 (EK1100)"}
    {attribute addProperty PreviousPort "Term 17 (EK1110) : B"}
    {attribute addProperty SyncUnit "default"}
    Term_18_EK1100 : Term_18_EK1100_20659A8D;
    {attribute addProperty Name "Term 23 (EK1100)"}
    {attribute addProperty PreviousPort "Term 10 (EK1122) : B"}
    {attribute addProperty SyncUnit "default"}
    Term_23_EK1100 : Term_23_EK1100_DFBF0BE4;
END_STRUCT
END_TYPE

// ---- DUTs/IO/Topology/Term_9_EK1100_91BFEC25.TcDUT
{attribute 'GeneratedUsingTerminal: EK1100-0000-0018'}
{attribute addProperty BoxType "EK1100-0000-0018"}
{attribute addProperty Id "Term_10_EK1122Term_10_EK1122_3D069EC11185Term_34_EL3403EL3403_812980A665Term_35_EL6001EL6001_0DE01E7E61Term_36_EL3024EL3024_C6E76B5A40Term_33_EL9011EL9011_D65D3D320"}
{attribute addProperty CRC "2445274149"}
{attribute addProperty Size "1351"}
{attribute addProperty Name "Term 9 (EK1100)"}
TYPE Term_9_EK1100_91BFEC25 EXTENDS EK1100_1FC0878B :
STRUCT
    {attribute addProperty Name "Term 10 (EK1122)"}
    {attribute addProperty PreviousPort "Term 9 (EK1100) : B"}
    {attribute addProperty SyncUnit "default"}
    Term_10_EK1122 : Term_10_EK1122_3D069EC1;
    {attribute addProperty Name "Term 34 (EL3403)"}
    {attribute addProperty PreviousPort "Term 10 (EK1122) : C"}
    {attribute addProperty SyncUnit "Row_0"}
    Term_34_EL3403 : EL3403_812980A6;
    {attribute addProperty Name "Term 35 (EL6001)"}
    {attribute addProperty PreviousPort "Term 34 (EL3403) : B"}
    {attribute addProperty SyncUnit "Row_0"}
    Term_35_EL6001 : EL6001_0DE01E7E;
    {attribute addProperty Name "Term 36 (EL3024)"}
    {attribute addProperty PreviousPort "Term 35 (EL6001) : B"}
    {attribute addProperty SyncUnit "Row_0"}
    Term_36_EL3024 : EL3024_C6E76B5A;
    {attribute addProperty Name "Term 33 (EL9011)"}
    {attribute addProperty PreviousPort "Term 36 (EL3024) : B"}
    {attribute addProperty SyncUnit "default"}
    Term_33_EL9011 : EL9011_D65D3D32;
END_STRUCT
END_TYPE

// ---- DUTs/IO/Topology/Device_2_EtherCAT_22CD061B.TcDUT
{attribute 'GeneratedUsingTerminal: IODEVICETYPE_ETHERCATPROT'}
{attribute addProperty BoxType "IODEVICETYPE_ETHERCATPROT"}
{attribute addProperty Id "Term_9_EK1100Term_9_EK1100_91BFEC251351SyncUnitsSyncUnits_F0D163CC108InputsInputs_A65FACA410OutputsOutputs_23C0ED1D6InfoDataInfoData_84133AC922"}
{attribute addProperty CRC "583861787"}
{attribute addProperty Size "1497"}
{attribute addProperty Name "Device 2 (EtherCAT)"}
TYPE Device_2_EtherCAT_22CD061B EXTENDS TcoIo.EtcMasterBase_62654B43 :
STRUCT
    {attribute addProperty Name "Term 9 (EK1100)"}
    {attribute addProperty PreviousPort "Device 2 (EtherCAT) : Master"}
    {attribute addProperty SyncUnit "default"}
    Term_9_EK1100 : Term_9_EK1100_91BFEC25;
    {attribute addProperty Name "SyncUnits"}
    SyncUnits : SyncUnits_F0D163CC;
    {attribute addProperty Name "Inputs"}
    Inputs : TcoIo.Inputs_A65FACA4;
    {attribute addProperty Name "Outputs"}
    Outputs : TcoIo.Outputs_23C0ED1D;
    {attribute addProperty Name "InfoData"}
    InfoData : TcoIo.InfoData_84133AC9;
END_STRUCT
END_TYPE

// ---- DUTs/IO/Topology/Term_157_EK1100_7C4BDD77.TcDUT
{attribute 'GeneratedUsingTerminal: EK1100-0000-0018'}
{attribute addProperty BoxType "EK1100-0000-0018"}
{attribute addProperty Id "Term_159_EL1809EL1809_32157CFD20"}
{attribute addProperty CRC "2085346679"}
{attribute addProperty Size "20"}
{attribute addProperty Name "Term 157 (EK1100)"}
TYPE Term_157_EK1100_7C4BDD77 EXTENDS EK1100_1FC0878B :
STRUCT
    {attribute addProperty Name "Term 159 (EL1809)"}
    {attribute addProperty PreviousPort "Term 157 (EK1100) : B"}
    {attribute addProperty SyncUnit "default"}
    Term_159_EL1809 : EL1809_32157CFD;
END_STRUCT
END_TYPE

// ---- DUTs/IO/Topology/Term_158_EK1100_E3D699B1.TcDUT
{attribute 'GeneratedUsingTerminal: EK1100-0000-0018'}
{attribute addProperty BoxType "EK1100-0000-0018"}
{attribute addProperty Id "Term_160_EL1809EL1809_32157CFD20"}
{attribute addProperty CRC "3822492081"}
{attribute addProperty Size "20"}
{attribute addProperty Name "Term 158 (EK1100)"}
TYPE Term_158_EK1100_E3D699B1 EXTENDS EK1100_1FC0878B :
STRUCT
    {attribute addProperty Name "Term 160 (EL1809)"}
    {attribute addProperty PreviousPort "Term 158 (EK1100) : B"}
    {attribute addProperty SyncUnit "default"}
    Term_160_EL1809 : EL1809_32157CFD;
END_STRUCT
END_TYPE

// ---- DUTs/IO/Topology/Term_154_EK1122_E57516AE.TcDUT
{attribute 'GeneratedUsingTerminal: EK1122-0000-0018'}
{attribute addProperty BoxType "EK1122-0000-0018"}
{attribute addProperty Id "Term_157_EK1100Term_157_EK1100_7C4BDD7720Term_158_EK1100Term_158_EK1100_E3D699B120"}
{attribute addProperty CRC "3849655982"}
{attribute addProperty Size "40"}
{attribute addProperty Name "Term 154 (EK1122)"}
TYPE Term_154_EK1122_E57516AE EXTENDS EK1122_1FC0878B :
STRUCT
    {attribute addProperty Name "Term 157 (EK1100)"}
    {attribute addProperty PreviousPort "Term 154 (EK1122) : D"}
    {attribute addProperty SyncUnit "default"}
    Term_157_EK1100 : Term_157_EK1100_7C4BDD77;
    {attribute addProperty Name "Term 158 (EK1100)"}
    {attribute addProperty PreviousPort "Term 154 (EK1122) : B"}
    {attribute addProperty SyncUnit "default"}
    Term_158_EK1100 : Term_158_EK1100_E3D699B1;
END_STRUCT
END_TYPE

// ---- DUTs/IO/Topology/Term_153_EK1100_91C0BB48.TcDUT
{attribute 'GeneratedUsingTerminal: EK1100-0000-0018'}
{attribute addProperty BoxType "EK1100-0000-0018"}
{attribute addProperty Id "Term_154_EK1122Term_154_EK1122_E57516AE40Term_155_EL2008EL2008_E2806B9511Term_156_EL2008EL2008_E2806B9511"}
{attribute addProperty CRC "2445327176"}
{attribute addProperty Size "62"}
{attribute addProperty Name "Term 153 (EK1100)"}
TYPE Term_153_EK1100_91C0BB48 EXTENDS EK1100_1FC0878B :
STRUCT
    {attribute addProperty Name "Term 154 (EK1122)"}
    {attribute addProperty PreviousPort "Term 153 (EK1100) : B"}
    {attribute addProperty SyncUnit "default"}
    Term_154_EK1122 : Term_154_EK1122_E57516AE;
    {attribute addProperty Name "Term 155 (EL2008)"}
    {attribute addProperty PreviousPort "Term 154 (EK1122) : C"}
    {attribute addProperty SyncUnit "default"}
    Term_155_EL2008 : EL2008_E2806B95;
    {attribute addProperty Name "Term 156 (EL2008)"}
    {attribute addProperty PreviousPort "Term 155 (EL2008) : B"}
    {attribute addProperty SyncUnit "default"}
    Term_156_EL2008 : EL2008_E2806B95;
END_STRUCT
END_TYPE

// ---- DUTs/IO/Topology/Term_180_EK1100_796B7783.TcDUT
{attribute 'GeneratedUsingTerminal: EK1100-0000-0018'}
{attribute addProperty BoxType "EK1100-0000-0018"}
{attribute addProperty Id "Term_181_EL1809EL1809_32157CFD20"}
{attribute addProperty CRC "2037086083"}
{attribute addProperty Size "20"}
{attribute addProperty Name "Term 180 (EK1100)"}
TYPE Term_180_EK1100_796B7783 EXTENDS EK1100_1FC0878B :
STRUCT
    {attribute addProperty Name "Term 181 (EL1809)"}
    {attribute addProperty PreviousPort "Term 180 (EK1100) : B"}
    {attribute addProperty SyncUnit "default"}
    Term_181_EL1809 : EL1809_32157CFD;
END_STRUCT
END_TYPE

// ---- DUTs/IO/Topology/Term_182_EK1100_E6B2C35E.TcDUT
{attribute 'GeneratedUsingTerminal: EK1100-0000-0018'}
{attribute addProperty BoxType "EK1100-0000-0018"}
{attribute addProperty Id "Term_183_EL1809EL1809_32157CFD20"}
{attribute addProperty CRC "3870475102"}
{attribute addProperty Size "20"}
{attribute addProperty Name "Term 182 (EK1100)"}
TYPE Term_182_EK1100_E6B2C35E EXTENDS EK1100_1FC0878B :
STRUCT
    {attribute addProperty Name "Term 183 (EL1809)"}
    {attribute addProperty PreviousPort "Term 182 (EK1100) : B"}
    {attribute addProperty SyncUnit "default"}
    Term_183_EL1809 : EL1809_32157CFD;
END_STRUCT
END_TYPE

// ---- DUTs/IO/Topology/Term_179_EK1122_2A33725A.TcDUT
{attribute 'GeneratedUsingTerminal: EK1122-0000-0018'}
{attribute addProperty BoxType "EK1122-0000-0018"}
{attribute addProperty Id "Term_180_EK1100Term_180_EK1100_796B778320Term_182_EK1100Term_182_EK1100_E6B2C35E20"}
{attribute addProperty CRC "708014682"}
{attribute addProperty Size "40"}
{attribute addProperty Name "Term 179 (EK1122)"}
TYPE Term_179_EK1122_2A33725A EXTENDS EK1122_1FC0878B :
STRUCT
    {attribute addProperty Name "Term 180 (EK1100)"}
    {attribute addProperty PreviousPort "Term 179 (EK1122) : D"}
    {attribute addProperty SyncUnit "default"}
    Term_180_EK1100 : Term_180_EK1100_796B7783;
    {attribute addProperty Name "Term 182 (EK1100)"}
    {attribute addProperty PreviousPort "Term 179 (EK1122) : B"}
    {attribute addProperty SyncUnit "default"}
    Term_182_EK1100 : Term_182_EK1100_E6B2C35E;
END_STRUCT
END_TYPE

// ---- DUTs/IO/Topology/Term_178_EK1100_9B7E9852.TcDUT
{attribute 'GeneratedUsingTerminal: EK1100-0000-0018'}
{attribute addProperty BoxType "EK1100-0000-0018"}
{attribute addProperty Id "Term_179_EK1122Term_179_EK1122_2A33725A40Term_184_EL2008EL2008_E2806B9511Term_185_EL2008EL2008_E2806B9511"}
{attribute addProperty CRC "2608765010"}
{attribute addProperty Size "62"}
{attribute addProperty Name "Term 178 (EK1100)"}
TYPE Term_178_EK1100_9B7E9852 EXTENDS EK1100_1FC0878B :
STRUCT
    {attribute addProperty Name "Term 179 (EK1122)"}
    {attribute addProperty PreviousPort "Term 178 (EK1100) : B"}
    {attribute addProperty SyncUnit "default"}
    Term_179_EK1122 : Term_179_EK1122_2A33725A;
    {attribute addProperty Name "Term 184 (EL2008)"}
    {attribute addProperty PreviousPort "Term 179 (EK1122) : C"}
    {attribute addProperty SyncUnit "default"}
    Term_184_EL2008 : EL2008_E2806B95;
    {attribute addProperty Name "Term 185 (EL2008)"}
    {attribute addProperty PreviousPort "Term 184 (EL2008) : B"}
    {attribute addProperty SyncUnit "default"}
    Term_185_EL2008 : EL2008_E2806B95;
END_STRUCT
END_TYPE

// ---- DUTs/IO/Topology/Term_147_EK1122_CA6A5D16.TcDUT
{attribute 'GeneratedUsingTerminal: EK1122-0000-0018'}
{attribute addProperty BoxType "EK1122-0000-0018"}
{attribute addProperty Id "Term_153_EK1100Term_153_EK1100_91C0BB4862Term_178_EK1100Term_178_EK1100_9B7E985262"}
{attribute addProperty CRC "3395968278"}
{attribute addProperty Size "124"}
{attribute addProperty Name "Term 147 (EK1122)"}
TYPE Term_147_EK1122_CA6A5D16 EXTENDS EK1122_1FC0878B :
STRUCT
    {attribute addProperty Name "Term 153 (EK1100)"}
    {attribute addProperty PreviousPort "Term 147 (EK1122) : D"}
    {attribute addProperty SyncUnit "default"}
    Term_153_EK1100 : Term_153_EK1100_91C0BB48;
    {attribute addProperty Name "Term 178 (EK1100)"}
    {attribute addProperty PreviousPort "Term 147 (EK1122) : B"}
    {attribute addProperty SyncUnit "default"}
    Term_178_EK1100 : Term_178_EK1100_9B7E9852;
END_STRUCT
END_TYPE

// ---- DUTs/IO/Topology/Term_189_EK1100_06A16014.TcDUT
{attribute 'GeneratedUsingTerminal: EK1100-0000-0018'}
{attribute addProperty BoxType "EK1100-0000-0018"}
{attribute addProperty Id "Term_193_EL1809EL1809_32157CFD20"}
{attribute addProperty CRC "111239188"}
{attribute addProperty Size "20"}
{attribute addProperty Name "Term 189 (EK1100)"}
TYPE Term_189_EK1100_06A16014 EXTENDS EK1100_1FC0878B :
STRUCT
    {attribute addProperty Name "Term 193 (EL1809)"}
    {attribute addProperty PreviousPort "Term 189 (EK1100) : B"}
    {attribute addProperty SyncUnit "default"}
    Term_193_EL1809 : EL1809_32157CFD;
END_STRUCT
END_TYPE

// ---- DUTs/IO/Topology/Term_194_EK1100_D4E2C05F.TcDUT
{attribute 'GeneratedUsingTerminal: EK1100-0000-0018'}
{attribute addProperty BoxType "EK1100-0000-0018"}
{attribute addProperty Id "Term_200_EL1809EL1809_32157CFD20"}
{attribute addProperty CRC "3571630175"}
{attribute addProperty Size "20"}
{attribute addProperty Name "Term 194 (EK1100)"}
TYPE Term_194_EK1100_D4E2C05F EXTENDS EK1100_1FC0878B :
STRUCT
    {attribute addProperty Name "Term 200 (EL1809)"}
    {attribute addProperty PreviousPort "Term 194 (EK1100) : B"}
    {attribute addProperty SyncUnit "default"}
    Term_200_EL1809 : EL1809_32157CFD;
END_STRUCT
END_TYPE

// ---- DUTs/IO/Topology/Term_188_EK1122_78D8AA43.TcDUT
{attribute 'GeneratedUsingTerminal: EK1122-0000-0018'}
{attribute addProperty BoxType "EK1122-0000-0018"}
{attribute addProperty Id "Term_189_EK1100Term_189_EK1100_06A1601420Term_194_EK1100Term_194_EK1100_D4E2C05F20"}
{attribute addProperty CRC "2027465283"}
{attribute addProperty Size "40"}
{attribute addProperty Name "Term 188 (EK1122)"}
TYPE Term_188_EK1122_78D8AA43 EXTENDS EK1122_1FC0878B :
STRUCT
    {attribute addProperty Name "Term 189 (EK1100)"}
    {attribute addProperty PreviousPort "Term 188 (EK1122) : D"}
    {attribute addProperty SyncUnit "default"}
    Term_189_EK1100 : Term_189_EK1100_06A16014;
    {attribute addProperty Name "Term 194 (EK1100)"}
    {attribute addProperty PreviousPort "Term 188 (EK1122) : B"}
    {attribute addProperty SyncUnit "default"}
    Term_194_EK1100 : Term_194_EK1100_D4E2C05F;
END_STRUCT
END_TYPE

// ---- DUTs/IO/Topology/Term_187_EK1100_648C31BD.TcDUT
{attribute 'GeneratedUsingTerminal: EK1100-0000-0018'}
{attribute addProperty BoxType "EK1100-0000-0018"}
{attribute addProperty Id "Term_188_EK1122Term_188_EK1122_78D8AA4340Term_204_EL2008EL2008_E2806B9511Term_205_EL2008EL2008_E2806B9511"}
{attribute addProperty CRC "1686909373"}
{attribute addProperty Size "62"}
{attribute addProperty Name "Term 187 (EK1100)"}
TYPE Term_187_EK1100_648C31BD EXTENDS EK1100_1FC0878B :
STRUCT
    {attribute addProperty Name "Term 188 (EK1122)"}
    {attribute addProperty PreviousPort "Term 187 (EK1100) : B"}
    {attribute addProperty SyncUnit "default"}
    Term_188_EK1122 : Term_188_EK1122_78D8AA43;
    {attribute addProperty Name "Term 204 (EL2008)"}
    {attribute addProperty PreviousPort "Term 188 (EK1122) : C"}
    {attribute addProperty SyncUnit "default"}
    Term_204_EL2008 : EL2008_E2806B95;
    {attribute addProperty Name "Term 205 (EL2008)"}
    {attribute addProperty PreviousPort "Term 204 (EL2008) : B"}
    {attribute addProperty SyncUnit "default"}
    Term_205_EL2008 : EL2008_E2806B95;
END_STRUCT
END_TYPE

// ---- DUTs/IO/Topology/Term_231_EK1100_6FCE8CEB.TcDUT
{attribute 'GeneratedUsingTerminal: EK1100-0000-0018'}
{attribute addProperty BoxType "EK1100-0000-0018"}
{attribute addProperty Id "Term_232_EL1809EL1809_32157CFD20"}
{attribute addProperty CRC "1875807467"}
{attribute addProperty Size "20"}
{attribute addProperty Name "Term 231 (EK1100)"}
TYPE Term_231_EK1100_6FCE8CEB EXTENDS EK1100_1FC0878B :
STRUCT
    {attribute addProperty Name "Term 232 (EL1809)"}
    {attribute addProperty PreviousPort "Term 231 (EK1100) : B"}
    {attribute addProperty SyncUnit "default"}
    Term_232_EL1809 : EL1809_32157CFD;
END_STRUCT
END_TYPE

// ---- DUTs/IO/Topology/Term_233_EK1100_CB654C3B.TcDUT
{attribute 'GeneratedUsingTerminal: EK1100-0000-0018'}
{attribute addProperty BoxType "EK1100-0000-0018"}
{attribute addProperty Id "Term_234_EL1809EL1809_32157CFD20"}
{attribute addProperty CRC "3412413499"}
{attribute addProperty Size "20"}
{attribute addProperty Name "Term 233 (EK1100)"}
TYPE Term_233_EK1100_CB654C3B EXTENDS EK1100_1FC0878B :
STRUCT
    {attribute addProperty Name "Term 234 (EL1809)"}
    {attribute addProperty PreviousPort "Term 233 (EK1100) : B"}
    {attribute addProperty SyncUnit "default"}
    Term_234_EL1809 : EL1809_32157CFD;
END_STRUCT
END_TYPE

// ---- DUTs/IO/Topology/Term_230_EK1122_16418046.TcDUT
{attribute 'GeneratedUsingTerminal: EK1122-0000-0018'}
{attribute addProperty BoxType "EK1122-0000-0018"}
{attribute addProperty Id "Term_231_EK1100Term_231_EK1100_6FCE8CEB20Term_233_EK1100Term_233_EK1100_CB654C3B20"}
{attribute addProperty CRC "373391430"}
{attribute addProperty Size "40"}
{attribute addProperty Name "Term 230 (EK1122)"}
TYPE Term_230_EK1122_16418046 EXTENDS EK1122_1FC0878B :
STRUCT
    {attribute addProperty Name "Term 231 (EK1100)"}
    {attribute addProperty PreviousPort "Term 230 (EK1122) : D"}
    {attribute addProperty SyncUnit "default"}
    Term_231_EK1100 : Term_231_EK1100_6FCE8CEB;
    {attribute addProperty Name "Term 233 (EK1100)"}
    {attribute addProperty PreviousPort "Term 230 (EK1122) : B"}
    {attribute addProperty SyncUnit "default"}
    Term_233_EK1100 : Term_233_EK1100_CB654C3B;
END_STRUCT
END_TYPE

// ---- DUTs/IO/Topology/Term_207_EK1100_2D36550A.TcDUT
{attribute 'GeneratedUsingTerminal: EK1100-0000-0018'}
{attribute addProperty BoxType "EK1100-0000-0018"}
{attribute addProperty Id "Term_230_EK1122Term_230_EK1122_1641804640Term_235_EL2008EL2008_E2806B9511Term_236_EL2008EL2008_E2806B9511"}
{attribute addProperty CRC "758535434"}
{attribute addProperty Size "62"}
{attribute addProperty Name "Term 207 (EK1100)"}
TYPE Term_207_EK1100_2D36550A EXTENDS EK1100_1FC0878B :
STRUCT
    {attribute addProperty Name "Term 230 (EK1122)"}
    {attribute addProperty PreviousPort "Term 207 (EK1100) : B"}
    {attribute addProperty SyncUnit "default"}
    Term_230_EK1122 : Term_230_EK1122_16418046;
    {attribute addProperty Name "Term 235 (EL2008)"}
    {attribute addProperty PreviousPort "Term 230 (EK1122) : C"}
    {attribute addProperty SyncUnit "default"}
    Term_235_EL2008 : EL2008_E2806B95;
    {attribute addProperty Name "Term 236 (EL2008)"}
    {attribute addProperty PreviousPort "Term 235 (EL2008) : B"}
    {attribute addProperty SyncUnit "default"}
    Term_236_EL2008 : EL2008_E2806B95;
END_STRUCT
END_TYPE

// ---- DUTs/IO/Topology/Term_186_EK1122_75C79D52.TcDUT
{attribute 'GeneratedUsingTerminal: EK1122-0000-0018'}
{attribute addProperty BoxType "EK1122-0000-0018"}
{attribute addProperty Id "Term_187_EK1100Term_187_EK1100_648C31BD62Term_207_EK1100Term_207_EK1100_2D36550A62"}
{attribute addProperty CRC "1976016210"}
{attribute addProperty Size "124"}
{attribute addProperty Name "Term 186 (EK1122)"}
TYPE Term_186_EK1122_75C79D52 EXTENDS EK1122_1FC0878B :
STRUCT
    {attribute addProperty Name "Term 187 (EK1100)"}
    {attribute addProperty PreviousPort "Term 186 (EK1122) : D"}
    {attribute addProperty SyncUnit "default"}
    Term_187_EK1100 : Term_187_EK1100_648C31BD;
    {attribute addProperty Name "Term 207 (EK1100)"}
    {attribute addProperty PreviousPort "Term 186 (EK1122) : B"}
    {attribute addProperty SyncUnit "default"}
    Term_207_EK1100 : Term_207_EK1100_2D36550A;
END_STRUCT
END_TYPE

// ---- DUTs/IO/Topology/Term_237_EK1122_86A8F7BD.TcDUT
{attribute 'GeneratedUsingTerminal: EK1122-0000-0018'}
{attribute addProperty BoxType "EK1122-0000-0018"}
{attribute addProperty Id "Drive_238_AX5101_0000_0214AX5101_1BD22F5129"}
{attribute addProperty CRC "2259220413"}
{attribute addProperty Size "29"}
{attribute addProperty Name "Term 237 (EK1122)"}
TYPE Term_237_EK1122_86A8F7BD EXTENDS EK1122_1FC0878B :
STRUCT
    {attribute addProperty Name "Drive 238 (AX5101-0000-0214)"}
    {attribute addProperty PreviousPort "Term 237 (EK1122) : D"}
    {attribute addProperty SyncUnit "default"}
    Drive_238_AX5101_0000_0214 : AX5101_1BD22F51;
END_STRUCT
END_TYPE

// ---- DUTs/IO/Topology/Term_289_EK1100_9C677E50.TcDUT
{attribute 'GeneratedUsingTerminal: EK1100-0000-0018'}
{attribute addProperty BoxType "EK1100-0000-0018"}
{attribute addProperty Id "Term_237_EK1122Term_237_EK1122_86A8F7BD29Term_293_EL1809EL1809_32157CFD20"}
{attribute addProperty CRC "2624028240"}
{attribute addProperty Size "49"}
{attribute addProperty Name "Term 289 (EK1100)"}
TYPE Term_289_EK1100_9C677E50 EXTENDS EK1100_1FC0878B :
STRUCT
    {attribute addProperty Name "Term 237 (EK1122)"}
    {attribute addProperty PreviousPort "Term 289 (EK1100) : B"}
    {attribute addProperty SyncUnit "default"}
    Term_237_EK1122 : Term_237_EK1122_86A8F7BD;
    {attribute addProperty Name "Term 293 (EL1809)"}
    {attribute addProperty PreviousPort "Term 237 (EK1122) : C"}
    {attribute addProperty SyncUnit "default"}
    Term_293_EL1809 : EL1809_32157CFD;
END_STRUCT
END_TYPE

